(* CODESYS project BASIC.library
   Company: OSCAT
   DefaultNamespace: OSCAT_BASIC
   LanguageModelAttribute: qualified-access-only
   Title: BASIC
   Description: OSCAT Library with basic POUs.
      see www.oscat.de home of OSCAT library
   Author: OSCAT
   Version: 3.3.3.0

Project tree, tasks and I/O mapping:
  libraries: Standard, 3.5.2.0 (System)
  Data types/
    data type CALENDAR
    data type COMPLEX
    data type CONSTANTS_LANGUAGE
    data type CONSTANTS_LOCATION
    data type CONSTANTS_MATH
    data type CONSTANTS_PHYS
    data type CONSTANTS_SETUP
    data type ESR_DATA
    data type FRACTION
    data type HOLIDAY_DATA
    data type REAL2
    data type SDT
    data type TIMER_EVENT
    data type VECTOR_3
  Global Variables/
    global variables Constants
    global variables Globale_Variablen
    global variables Setup_Data
  POUs/
    Buffer Management/
      function _BUFFER_CLEAR [ST]
      function _BUFFER_INIT [ST]
      function _BUFFER_INSERT [ST]
      function _BUFFER_UPPERCASE [ST]
      function _STRING_TO_BUFFER [ST]
      function BUFFER_COMP [ST]
      function BUFFER_SEARCH [ST]
      function BUFFER_TO_STRING [ST]
    Engineering/
      automation/
        function block DRIVER_1 [ST]
        function block DRIVER_4 [ST]
        function block DRIVER_4C [ST]
        function block FLOW_CONTROL [ST]
        function block FT_Profile [ST]
        function block INC_DEC [ST]
        function block INTERLOCK [ST]
        function block INTERLOCK_4 [ST]
        function MANUAL [ST]
        function block MANUAL_1 [ST]
        function block MANUAL_2 [ST]
        function block MANUAL_4 [ST]
        function block PARSET [ST]
        function block PARSET2 [ST]
        function block SIGNAL [ST]
        function block SIGNAL_4 [ST]
        function block SRAMP [ST]
        function block TUNE [ST]
        function block TUNE2 [ST]
      control/
        function BAND_B [ST]
        function block CONTROL_SET1 [ST]
        function block CONTROL_SET2 [ST]
        function CTRL_IN [ST]
        function block CTRL_OUT [ST]
        function block CTRL_PI [ST]
        function block CTRL_PID [ST]
        function block CTRL_PWM [ST]
        function DEAD_BAND [ST]
        function block DEAD_BAND_A [ST]
        function DEAD_ZONE [ST]
        function block DEAD_ZONE2 [ST]
        function block FT_DERIV [ST]
        function block FT_IMP [ST]
        function block FT_INT [ST]
        function block FT_INT2 [ST]
        function block FT_PD [ST]
        function block FT_PDT1 [ST]
        function block FT_PI [ST]
        function block FT_PID [ST]
        function block FT_PIDW [ST]
        function block FT_PIDWL [ST]
        function block FT_PIW [ST]
        function block FT_PIWL [ST]
        function block FT_PT1 [ST]
        function block FT_PT2 [ST]
        function block FT_TN16 [ST]
        function block FT_TN64 [ST]
        function block FT_TN8 [ST]
        function block HYST [ST]
        function block HYST_1 [ST]
        function block HYST_2 [ST]
        function block HYST_3 [ST]
        function block INTEGRATE [ST]
      conversion/
        function block ASTRO [ST]
        function BFT_TO_MS [ST]
        function C_TO_F [ST]
        function C_TO_K [ST]
        function DEG_TO_DIR [ST]
        function DIR_TO_DEG [ST]
        function block ENERGY [ST]
        function F_TO_C [ST]
        function F_TO_OM [ST]
        function F_TO_PT [ST]
        function GEO_TO_DEG [ST]
        function K_TO_C [ST]
        function KMH_TO_MS [ST]
        function block LENGTH [ST]
        function MS_TO_BFT [ST]
        function MS_TO_KMH [ST]
        function OM_TO_F [ST]
        function block PRESSURE [ST]
        function PT_TO_F [ST]
        function block SPEED [ST]
        function block TEMPERATURE [ST]
      measurements/
        function block ALARM_2 [ST]
        function block BAR_GRAPH [ST]
        function block CALIBRATE [ST]
        function block CYCLE_TIME [ST]
        function block DT_SIMU [ST]
        function block FLOW_METER [ST]
        function block M_D [ST]
        function block M_T [ST]
        function block M_TX [ST]
        function block METER [ST]
        function block METER_STAT [ST]
        function block ONTIME [ST]
        function T_PLC_MS [ST]
        function T_PLC_US [ST]
        function block TC_MS [ST]
        function block TC_S [ST]
        function block TC_US [ST]
      sensor/
        function MULTI_IN [ST]
        function RES_NI [ST]
        function RES_NTC [ST]
        function RES_PT [ST]
        function RES_SI [ST]
        function SENSOR_INT [ST]
        function TEMP_NI [ST]
        function TEMP_NTC [ST]
        function TEMP_PT [ST]
        function TEMP_SI [ST]
      signal generators/
        function block _RMP_B [ST]
        function block _RMP_NEXT [ST]
        function block _RMP_W [ST]
        function block GEN_PULSE [ST]
        function block GEN_PW2 [ST]
        function block GEN_RDM [ST]
        function block GEN_RDT [ST]
        function block GEN_RMP [ST]
        function block GEN_SIN [ST]
        function block GEN_SQR [ST]
        function block PWM_DC [ST]
        function block PWM_PW [ST]
        function block RMP_B [ST]
        function block RMP_SOFT [ST]
        function block RMP_W [ST]
      signal processing/
        function AIN [ST]
        function block AIN1 [ST]
        function AOUT [ST]
        function AOUT1 [ST]
        function BYTE_TO_RANGE [ST]
        function block DELAY [ST]
        function block DELAY_4 [ST]
        function block FADE [ST]
        function block FILTER_DW [ST]
        function block FILTER_I [ST]
        function block FILTER_MAV_DW [ST]
        function block FILTER_MAV_W [ST]
        function block FILTER_W [ST]
        function block FILTER_WAV [ST]
        function MIX [ST]
        function MUX_R2 [ST]
        function MUX_R4 [ST]
        function OFFSET [ST]
        function OFFSET2 [ST]
        function OVERRIDE [ST]
        function RANGE_TO_BYTE [ST]
        function RANGE_TO_WORD [ST]
        function SCALE [ST]
        function SCALE_B [ST]
        function SCALE_B2 [ST]
        function SCALE_B4 [ST]
        function SCALE_B8 [ST]
        function SCALE_D [ST]
        function SCALE_R [ST]
        function SCALE_X2 [ST]
        function SCALE_X4 [ST]
        function SCALE_X8 [ST]
        function block SEL2_OF_3 [ST]
        function block SEL2_OF_3B [ST]
        function block SH [ST]
        function block SH_1 [ST]
        function block SH_2 [ST]
        function block SH_T [ST]
        function STAIR [ST]
        function block STAIR2 [ST]
        function block TREND [ST]
        function block TREND_DW [ST]
        function WORD_TO_RANGE [ST]
    List Processing/
      function LIST_ADD [ST]
      function LIST_CLEAN [ST]
      function LIST_GET [ST]
      function LIST_INSERT [ST]
      function LIST_LEN [ST]
      function block LIST_NEXT [ST]
      function LIST_RETRIEVE [ST]
      function LIST_RETRIEVE_LAST [ST]
    Logic/
      FF edge triggered/
        function block COUNT_BR [ST]
        function block COUNT_DR [ST]
        function block FF_D2E [ST]
        function block FF_D4E [ST]
        function block FF_DRE [ST]
        function block FF_JKE [ST]
        function block FF_RSE [ST]
        function block SELECT_8 [ST]
        function block SHR_4E [ST]
        function block SHR_4UDE [ST]
        function block SHR_8PLE [ST]
        function block SHR_8UDE [ST]
        function block TOGGLE [ST]
      FF pulse triggered/
        function block LTCH [ST]
        function block LTCH_4 [ST]
        function block STORE_8 [ST]
      gate logic/
        function BCDC_TO_INT [ST]
        function BIT_COUNT [ST]
        function BIT_LOAD_B [ST]
        function BIT_LOAD_B2 [ST]
        function BIT_LOAD_DW [ST]
        function BIT_LOAD_DW2 [ST]
        function BIT_LOAD_W [ST]
        function BIT_LOAD_W2 [ST]
        function BIT_OF_DWORD [ST]
        function BIT_TOGGLE_B [ST]
        function BIT_TOGGLE_DW [ST]
        function BIT_TOGGLE_W [ST]
        function BYTE_OF_BIT [ST]
        function BYTE_OF_DWORD [ST]
        function block BYTE_TO_BITS [ST]
        function BYTE_TO_GRAY [ST]
        function CHECK_PARITY [ST]
        function CHK_REAL [ST]
        function block DEC_2 [ST]
        function block DEC_4 [ST]
        function block DEC_8 [ST]
        function DW_TO_REAL [ST]
        function DWORD_OF_BYTE [ST]
        function DWORD_OF_WORD [ST]
        function GRAY_TO_BYTE [ST]
        function INT_TO_BCDC [ST]
        function MUX_2 [ST]
        function MUX_4 [ST]
        function PARITY [ST]
        function REAL_TO_DW [ST]
        function REFLECT [ST]
        function REVERSE [ST]
        function SHL1 [ST]
        function SHR1 [ST]
        function SWAP_BYTE [ST]
        function SWAP_BYTE2 [ST]
        function WORD_OF_BYTE [ST]
        function WORD_OF_DWORD [ST]
      generators/
        function block A_TRIG [ST]
        function block B_TRIG [ST]
        function block CLICK_CNT [ST]
        function block CLICK_DEC [ST]
        function block CLK_DIV [ST]
        function block CLK_N [ST]
        function block CLK_PRG [ST]
        function block CLK_PULSE [ST]
        function block CYCLE_4 [ST]
        function block D_TRIG [ST]
        function block GEN_BIT [ST]
        function block GEN_SQ [ST]
        function block SCHEDULER [ST]
        function block SCHEDULER_2 [ST]
        function block SEQUENCE_4 [ST]
        function block SEQUENCE_64 [ST]
        function block SEQUENCE_8 [ST]
        function block TMAX [ST]
        function block TMIN [ST]
        function block TOF_1 [ST]
        function block TONOF [ST]
        function block TP_1 [ST]
        function block TP_1D [ST]
        function block TP_X [ST]
      memory/
        function block FIFO_16 [ST]
        function block FIFO_32 [ST]
        function block STACK_16 [ST]
        function block STACK_32 [ST]
      Others/
        function CRC_GEN [ST]
        function block MATRIX [ST]
        function block PIN_CODE [ST]
    Mathematical/
      Array/
        function _ARRAY_ABS [ST]
        function _ARRAY_ADD [ST]
        function _ARRAY_INIT [ST]
        function _ARRAY_MEDIAN [ST]
        function _ARRAY_MUL [ST]
        function _ARRAY_SHUFFLE [ST]
        function _ARRAY_SORT [ST]
        function ARRAY_AVG [ST]
        function ARRAY_GAV [ST]
        function ARRAY_HAV [ST]
        function ARRAY_MAX [ST]
        function ARRAY_MIN [ST]
        function ARRAY_SDV [ST]
        function ARRAY_SPR [ST]
        function ARRAY_SUM [ST]
        function ARRAY_TREND [ST]
        function ARRAY_VAR [ST]
        function IS_SORTED [ST]
      Complex/
        function CABS [ST]
        function CACOS [ST]
        function CACOSH [ST]
        function CADD [ST]
        function CARG [ST]
        function CASIN [ST]
        function CASINH [ST]
        function CATAN [ST]
        function CATANH [ST]
        function CCON [ST]
        function CCOS [ST]
        function CCOSH [ST]
        function CDIV [ST]
        function CEXP [ST]
        function CINV [ST]
        function CLOG [ST]
        function CMUL [ST]
        function CPOL [ST]
        function CPOW [ST]
        function CSET [ST]
        function CSIN [ST]
        function CSINH [ST]
        function CSQRT [ST]
        function CSUB [ST]
        function CTAN [ST]
        function CTANH [ST]
      Double Precision/
        function R2_ABS [ST]
        function R2_ADD [ST]
        function R2_ADD2 [ST]
        function R2_MUL [ST]
        function R2_SET [ST]
      functions/
        function F_LIN [ST]
        function F_LIN2 [ST]
        function F_POLY [ST]
        function F_POWER [ST]
        function F_QUAD [ST]
        function FRMP_B [ST]
        function block FT_AVG [ST]
        function block FT_MIN_MAX [ST]
        function block FT_RMP [ST]
        function LINEAR_INT [ST]
        function POLYNOM_INT [ST]
      Geometry/
        function CIRCLE_A [ST]
        function CIRCLE_C [ST]
        function CIRCLE_SEG [ST]
        function CONE_V [ST]
        function ELLIPSE_A [ST]
        function ELLIPSE_C [ST]
        function SPHERE_V [ST]
        function TRIANGLE_A [ST]
      Vektormathematik/
        function V3_ABS [ST]
        function V3_ADD [ST]
        function V3_ANG [ST]
        function V3_DPRO [ST]
        function V3_NORM [ST]
        function V3_NUL [ST]
        function V3_PAR [ST]
        function V3_REV [ST]
        function V3_SMUL [ST]
        function V3_SUB [ST]
        function V3_XANG [ST]
        function V3_XPRO [ST]
        function V3_YANG [ST]
        function V3_ZANG [ST]
      function ACOSH [ST]
      function ACOTH [ST]
      function AGDF [ST]
      function ASINH [ST]
      function ATAN2 [ST]
      function ATANH [ST]
      function BETA [ST]
      function BINOM [ST]
      function CAUCHY [ST]
      function CAUCHYCD [ST]
      function CEIL [ST]
      function CEIL2 [ST]
      function CMP [ST]
      function COSH [ST]
      function COTH [ST]
      function D_TRUNC [ST]
      function DEC1 [ST]
      function DEG [ST]
      function DIFFER [ST]
      function ERF [ST]
      function ERFC [ST]
      function EVEN [ST]
      function EXP10 [ST]
      function EXPN [ST]
      function FACT [ST]
      function FIB [ST]
      function FLOOR [ST]
      function FLOOR2 [ST]
      function FRACT [ST]
      function GAMMA [ST]
      function GAUSS [ST]
      function GAUSSCD [ST]
      function GCD [ST]
      function GDF [ST]
      function GOLD [ST]
      function HYPOT [ST]
      function INC [ST]
      function INC1 [ST]
      function INC2 [ST]
      function INV [ST]
      function LAMBERT_W [ST]
      function LANGEVIN [ST]
      function MAX3 [ST]
      function MID3 [ST]
      function MIN3 [ST]
      function MODR [ST]
      function MUL_ADD [ST]
      function NEGX [ST]
      function RAD [ST]
      function RDM [ST]
      function RDM2 [ST]
      function RDMDW [ST]
      function REAL_TO_FRAC [ST]
      function RND [ST]
      function ROUND [ST]
      function SGN [ST]
      function SIGMOID [ST]
      function SIGN_I [ST]
      function SIGN_R [ST]
      function SINC [ST]
      function SINH [ST]
      function SQRTN [ST]
      function TANC [ST]
      function TANH [ST]
      function WINDOW [ST]
      function WINDOW2 [ST]
    Other/
      function block ESR_COLLECT [ST]
      function block ESR_MON_B8 [ST]
      function block ESR_MON_R4 [ST]
      function block ESR_MON_X8 [ST]
      function OSCAT_VERSION [ST]
      function STATUS_TO_ESR [ST]
    String/
      function BIN_TO_BYTE [ST]
      function BIN_TO_DWORD [ST]
      function BYTE_TO_STRB [ST]
      function BYTE_TO_STRH [ST]
      function CAPITALIZE [ST]
      function CHARCODE [ST]
      function CHARNAME [ST]
      function CHR_TO_STRING [ST]
      function CLEAN [ST]
      function CODE [ST]
      function COUNT_CHAR [ST]
      function COUNT_SUBSTRING [ST]
      function DEC_TO_BYTE [ST]
      function DEC_TO_DWORD [ST]
      function DEC_TO_INT [ST]
      function DEL_CHARS [ST]
      function DT_TO_STRF [ST]
      function DWORD_TO_STRB [ST]
      function DWORD_TO_STRF [ST]
      function DWORD_TO_STRH [ST]
      function EXEC [ST]
      function FILL [ST]
      function FIND_CHAR [ST]
      function FIND_CTRL [ST]
      function FIND_NONUM [ST]
      function FIND_NUM [ST]
      function FINDB [ST]
      function FINDB_NONUM [ST]
      function FINDB_NUM [ST]
      function FINDP [ST]
      function FIX [ST]
      function FLOAT_TO_REAL [ST]
      function FSTRING_TO_BYTE [ST]
      function FSTRING_TO_DT [ST]
      function FSTRING_TO_DWORD [ST]
      function FSTRING_TO_MONTH [ST]
      function FSTRING_TO_WEEK [ST]
      function FSTRING_TO_WEEKDAY [ST]
      function HEX_TO_BYTE [ST]
      function HEX_TO_DWORD [ST]
      function IS_ALNUM [ST]
      function IS_ALPHA [ST]
      function IS_CC [ST]
      function IS_CTRL [ST]
      function IS_HEX [ST]
      function IS_LOWER [ST]
      function IS_NCC [ST]
      function IS_NUM [ST]
      function IS_UPPER [ST]
      function ISC_ALPHA [ST]
      function ISC_CTRL [ST]
      function ISC_HEX [ST]
      function ISC_LOWER [ST]
      function ISC_NUM [ST]
      function ISC_UPPER [ST]
      function LOWERCASE [ST]
      function block MESSAGE_4R [ST]
      function block MESSAGE_8 [ST]
      function MIRROR [ST]
      function MONTH_TO_STRING [ST]
      function OCT_TO_BYTE [ST]
      function OCT_TO_DWORD [ST]
      function REAL_TO_STRF [ST]
      function REPLACE_ALL [ST]
      function REPLACE_CHARS [ST]
      function REPLACE_UML [ST]
      function block TICKER [ST]
      function TO_LOWER [ST]
      function TO_UML [ST]
      function TO_UPPER [ST]
      function TRIM [ST]
      function TRIM1 [ST]
      function TRIME [ST]
      function UPPERCASE [ST]
      function WEEKDAY_TO_STRING [ST]
      function LREAL_TO_STRF [ST]
    Time&Date/
      function block CALENDAR_CALC [ST]
      function DATE_ADD [ST]
      function DAY_OF_DATE [ST]
      function DAY_OF_MONTH [ST]
      function DAY_OF_WEEK [ST]
      function DAY_OF_YEAR [ST]
      function DAY_TO_TIME [ST]
      function DAYS_DELTA [ST]
      function DAYS_IN_MONTH [ST]
      function DAYS_IN_YEAR [ST]
      function block DCF77 [ST]
      function DST [ST]
      function DT2_TO_SDT [ST]
      function DT_TO_SDT [ST]
      function EASTER [ST]
      function block EVENTS [ST]
      function block HOLIDAY [ST]
      function HOUR [ST]
      function HOUR_OF_DT [ST]
      function HOUR_TO_TIME [ST]
      function HOUR_TO_TOD [ST]
      function JD2000 [ST]
      function LEAP_DAY [ST]
      function LEAP_OF_DATE [ST]
      function LEAP_YEAR [ST]
      function LTIME_TO_UTC [ST]
      function MINUTE [ST]
      function MINUTE_OF_DT [ST]
      function MINUTE_TO_TIME [ST]
      function MONTH_BEGIN [ST]
      function MONTH_END [ST]
      function MONTH_OF_DATE [ST]
      function MULTIME [ST]
      function PERIOD [ST]
      function PERIOD2 [ST]
      function REFRACTION [ST]
      function block RTC_2 [ST]
      function block RTC_MS [ST]
      function SDT_TO_DATE [ST]
      function SDT_TO_DT [ST]
      function SDT_TO_TOD [ST]
      function SECOND [ST]
      function SECOND_OF_DT [ST]
      function SECOND_TO_TIME [ST]
      function SET_DATE [ST]
      function SET_DT [ST]
      function SET_TOD [ST]
      function SUN_MIDDAY [ST]
      function block SUN_POS [ST]
      function block SUN_TIME [ST]
      function TIMECHECK [ST]
      function UTC_TO_LTIME [ST]
      function WORK_WEEK [ST]
      function YEAR_BEGIN [ST]
      function YEAR_END [ST]
      function YEAR_OF_DATE [ST]
*)

// Data types/CALENDAR
TYPE CALENDAR :
STRUCT
	UTC : DT;					(* world time UTC *)
	_LDT : DT;					(* local time *)
	_LDATE : DATE;				(* local date *)
	_LTOD : TOD;					(* local time of day *)
	YEAR : INT;					(* year of LDATE *)
	MONTH : INT;				(* month of LDATE *)
	DAY : INT;					(* day of LDATE *)
	WEEKDAY : INT;				(* weekday of LDATE *)
	OFFSET : INT;				(* Time Zone Offset for Local time in minutes *)
	DST_EN : BOOL;				(* daylight savings time enable *)
	DST_ON : BOOL;				(* true when daylight savings time os on *)
	NAME : STRING(5);			(* name of time zone *)
	LANGUAGE : INT;			(* location number pls see location setup *)
	LONGITUDE : REAL;			(* longitude of current location *)
	LATITUDE : REAL;			(* latitude of current location *)
	SUN_RISE : TOD;				(* sun_rise for current location *)
	SUN_SET : TOD;				(* sun_set for current location *)
	SUN_MIDDAY : TOD;			(* worldtime when sun stands at south position *)
	SUN_HEIGTH : REAL	;		(* suns heigth at midday, south position *)
	SUN_HOR : REAL;			(* sun angle horizontal 0 = north in degrees *)
	SUN_VER : REAL;			(* sun angle vertical above horizon in degrees *)
	NIGHT : BOOL;				(* true between sun_set and sun_rise *)
	HOLIDAY : BOOL;			(* true when holiday *)
	HOLY_NAME : STRING(30);	(* name of holiday *)
	WORK_WEEK : INT;			(* current work week *)
END_STRUCT
END_TYPE

// Data types/COMPLEX
TYPE COMPLEX :
STRUCT
	re : REAL;
	im : REAL;
END_STRUCT
END_TYPE

// Data types/CONSTANTS_LANGUAGE
TYPE CONSTANTS_LANGUAGE :
STRUCT
	(* Language Setup *)
	DEFAULT : INT := 1; (* 1=english, 2=german 3=french *)
	LMAX : INT := 3;
	WEEKDAYS : ARRAY[1..3, 1..7] OF STRING(10) :=[	'Monday', 'Tuesday', 'Wednesday', 'Thursday', 'Friday', 'Saturday', 'Sunday',
													'Montag', 'Dienstag', 'Mittwoch', 'Donnerstag', 'Freitag', 'Samstag', 'Sonntag',
													'Lundi', 'Mardi', 'Mercredi', 'Jeudi', 'Vendredi', 'Samedi', 'Dimanche'];
	WEEKDAYS2 : ARRAY[1..3, 1..7] OF STRING(2) :=[	'Mo', 'Tu', 'We', 'Th', 'Fr', 'Sa', 'Su',
													'Mo', 'Di', 'Mi', 'Do', 'Fr', 'Sa', 'So',
													'Lu', 'Ma', 'Me', 'Je', 'Ve', 'Sa', 'Di'];
	MONTHS : ARRAY[1..3, 1..12] OF STRING(10) :=[	'January', 'February', 'March', 'April', 'May', 'June', 'July', 'August', 'September', 'October', 'November', 'December',
													'Januar', 'Februar', 'März', 'April', 'Mai', 'Juni', 'Juli', 'August', 'September', 'Oktober', 'November', 'Dezember',
													'Janvier', 'Février', 'mars', 'Avril', 'Mai', 'Juin', 'Juillet', 'Août', 'Septembre', 'Octobre', 'Novembre', 'Decembre'];
	MONTHS3 : ARRAY[1..3, 1..12] OF STRING(3) :=[	'Jan', 'Feb', 'Mar', 'Apr', 'May', 'Jun', 'Jul', 'Aug', 'Sep', 'Oct', 'Nov', 'Dec',
													'Jan', 'Feb', 'Mrz', 'Apr', 'Mai', 'Jun', 'Jul', 'Aug', 'Sep', 'Okt', 'Nov', 'Dez',
													'Jan', 'Fev', 'Mar', 'Avr', 'Mai', 'Jun', 'Jul', 'Aou', 'Sep', 'Oct', 'Nov', 'Dec'];
	DIRS : ARRAY[1..3,0..15] OF STRING(3) :=[		'N', 'NNE', 'NE', 'ENE', 'E', 'ESE', 'SE', 'SSE', 'S', 'SSW', 'SW', 'WSW', 'W', 'WNW', 'NW', 'NNW',
													'N', 'NNO', 'NO', 'ONO', 'O', 'OSO', 'SO', 'SSO', 'S', 'SSW', 'SW', 'WSW', 'W', 'WNW', 'NW', 'NNW',
													'N', 'NNO', 'NO', 'ONO', 'O', 'OSO', 'SO', 'SSO', 'S', 'SSW', 'SW', 'WSW', 'W', 'WNW', 'NW', 'NNW'];
END_STRUCT
END_TYPE

// Data types/CONSTANTS_LOCATION
TYPE CONSTANTS_LOCATION :
STRUCT
	(* location setup *)
	DEFAULT : INT := 1; (* 1=germany, 2=austria 3=france 4=belgium-german 5= italien-Südtirol *)
	LMAX : INT := 5;

	(* language spoken in the location *)
	LANGUAGE : ARRAY[1..5] OF INT :=[ 2, 2, 3, 2, 2];

END_STRUCT
END_TYPE

// Data types/CONSTANTS_MATH
TYPE CONSTANTS_MATH :
STRUCT
	PI : REAL := 	3.14159265358979323846264338327950288;		(* Kreiszahl PI *)
	PI2 : REAL := 	6.28318530717958647692528676655900576;	(* PI * 2 *)
	PI4 : REAL :=  12.56637061435917295385057353311801152;	(* PI * 4 *)
	PI05 : REAL :=  1.5707963267949;							(* PI / 2 *)
	PI025 : REAL := 0.785398163397448;							(* PI / 4 *)
	PI_INV : REAL := 0.318309886183791;						(* 1 / PI *)
	E : REAL := 	2.71828182845904523536028747135266249;		(* Euler constant e *)
	E_INV : REAL := 0.367879441171442;							(* 1 / e *)
	SQ2 : REAL :=	1.4142135623731;							(* Wurzel von 2 *)
	FACTS : ARRAY[0..12] OF DINT :=[ 1,1,2,6,24,120,720,5040,40320,362880,3628800,39916800,479001600];
END_STRUCT
END_TYPE

// Data types/CONSTANTS_PHYS
TYPE CONSTANTS_PHYS :
STRUCT
	C : REAL := 299792458.0;				(* Lichtgeschwindigkeit in m/s *)
	E : REAL := 1.60217653E-19;				(* elementarladung in Colomb = A * s *)
	G : REAL := 9.80665; 						(* Erdbeschleunigung in m / s² *)
	T0 : REAL := -273.15;						(* absoluter Nullpunkt in °C *)
	RU : REAL := 8.314472; 					(* Universelle Gaskonstante in J / (mol · K) *)
	PN : REAL := 101325.0;					(* NormalDruck in Pa *)
END_STRUCT
END_TYPE

// Data types/CONSTANTS_SETUP
TYPE CONSTANTS_SETUP :
STRUCT
	(* setup Parameters *)
	EXTENDED_ASCII : BOOL := TRUE;
	CHARNAMES : ARRAY[1..4] OF STRING(253) :=[ ';"&quot;&&amp;<&lt;>&gt;€&euro; &nbsp;¡&iexcl;¢&cent;£&pound;¤&curren;¥&yen;¦&brvbar;§&sect;¨&uml;©&copy;ª&ordf;«&laquo;¬&not;­&shy;®&reg;¯&macr;°&deg;±&plusmn;²&sup2;³&sup3;´&acute;µ&micro;¶&para;·&middot;¸&cedil;¹&sup1;º&ordm;»&raquo;¼&frac14;Û&Ucirc;',
		';¾&frac34;¿&iquest;À&Agrave;Á&Aacute;Â&Acirc;Ã&Atilde;Ä&Auml;Å&Aring;Æ&AElig;Ç&Ccedil;È&Egrave;É&Eacute;Ê&Ecirc;Ë&Euml;Ì&Igrave;Í&Iacute;Î&Icirc;Ï&Iuml;Ð&ETH;Ñ&Ntilde;Ò&Ograve;Ó&Oacute;Ô&Ocirc;Õ&Otilde;Ö&Ouml;×&times;Ø&Oslash;Ù&Ugrave;Ú&Uacute;½&frac12;',
		';Ü&Uuml;Ý&Yacute;Þ&THORN;ß&szlig;à&agrave;á&aacute;â&acirc;ã&atilde;ä&auml;å&aring;æ&aelig;ç&ccedil;è&egrave;é&eacute;ê&ecirc;ë&euml;ì&igrave;í&iacute;î&icirc;ï&iuml;ð&eth;ñ&ntilde;ò&ograve;ó&oacute;ô&ocirc;õ&otilde;ö&ouml;÷&divide;ø&oslash;ù&ugrave;',
		';ú&uacute;û&ucirc;ü&uuml;ý&yacute;þ&thorn;ÿ&yuml;'];
	MTH_OFS : ARRAY[1..12] OF INT :=[ 0,31,59,90,120,151,181,212,243,273,304,334];
	DECADES : ARRAY[0..8] OF REAL :=[ 1.0,10.0,100.0,1000.0,10000.0,10000.0,100000.0,1000000.0,10000000.0];
END_STRUCT
END_TYPE

// Data types/ESR_DATA
TYPE ESR_DATA :
STRUCT
	TYP : BYTE;
	ADRESS : STRING(10);
	DS : DT;
	TS : TIME;
	DATA : ARRAY[0..7] OF BYTE;
END_STRUCT
END_TYPE

// Data types/FRACTION
TYPE FRACTION :
STRUCT
	NUMERATOR : INT;
	DENOMINATOR : INT;
END_STRUCT
END_TYPE

// Data types/HOLIDAY_DATA
TYPE HOLIDAY_DATA :
STRUCT
	NAME : STRING(30);
	DAY : SINT;
	MONTH : SINT;
	USE : SINT;
END_STRUCT
END_TYPE

// Data types/REAL2
TYPE REAL2 :
STRUCT
	R1 : REAL;	(* small value *)
	RX : REAL;	(* big value *)
END_STRUCT
END_TYPE

// Data types/SDT
TYPE SDT :
STRUCT
	YEAR : INT;
	MONTH : INT;
	DAY : INT;
	WEEKDAY : INT;
	HOUR : INT;
	MINUTE : INT;
	SECOND : INT;
	MS : INT;
END_STRUCT
END_TYPE

// Data types/TIMER_EVENT
TYPE TIMER_EVENT :
STRUCT
	TYP : BYTE;
	CHANNEL : BYTE;
	DAY : BYTE;
	START : TOD;
	DURATION : TIME;
	LAND : BYTE;
	LOR : BYTE;
	LAST : DT;
END_STRUCT
END_TYPE

// Data types/VECTOR_3
TYPE VECTOR_3 :
STRUCT
	X : REAL;
	Y : REAL;
	Z : REAL;
END_STRUCT
END_TYPE

// Global Variables/Constants
VAR_GLOBAL CONSTANT
	STRING_LENGTH : INT := 250;
	LIST_LENGTH : INT := 250;
END_VAR




(* revisionhistory
hm 3. mar. 2007
	extended accuracy of pi2
	renamed T0 to Tk for better compatibility with other libraries
	renamed C t0 c0 for better compatibility

hm	2. may. 2007
	added RU universal gas constant

hm	1. oct. 2007
	added setup parameter STEP7

hm 31. oct. 2007
	added PN

hm	6. mar. 2008
	added setup Parameter EXTENDED_ASCII

hm	28. Mar. 2008
	added setup parameter STRING_LENGTH

hm	7. apr. 2008
	Deleted unused setup parameter Step7

hm	19. apr. 2008
	added setup parameter NETWORK_BUFFER_SIZE

hm	27. apr. 2008
	added PI05 and PI025

hm	18. may. 2008
	added charname lists
	renamed E to E1

hm	30. jun. 2008
	reduced size of string constants to 253 to avoid problems with target aixia DCUF

hm	21. sep. 2008
	added section language setup
	added section location setup

hm	20. oct. 2008
	changed to structured constants

hm	16. nov. 2008
	moved structured constants to global vars for compatibility reasons

hm	13. nov. 2009
	added network_buffer_short_size
	renamed network_buffer_long_size
	changed string length to 250

hm	20. jan. 2011
	removed network buffers
	added list_length
*)

// Global Variables/Globale_Variablen
VAR_GLOBAL
	MATH : CONSTANTS_MATH;
	PHYS : CONSTANTS_PHYS;
	LANGUAGE : CONSTANTS_LANGUAGE;
	SETUP : CONSTANTS_SETUP;
	LOCATION : CONSTANTS_LOCATION;
END_VAR

// Global Variables/Setup_Data
VAR_GLOBAL RETAIN

END_VAR

// POUs/Mathematical/Array/_ARRAY_ABS
FUNCTION _ARRAY_ABS : BOOL
VAR_INPUT
	pt : POINTER TO ARRAY[0..32000] OF REAL;
	size : UINT;
END_VAR
VAR
	i: UINT;
	stop: UINT;
END_VAR

(*
version 1.0	2. apr. 2008
programmer 	hugo
tested by	tobias

this function will calculate the absolute value of each element of the array and stroe the result instead of the element.
Array[i] := ABS(ARRAY[i]).
the function needs to be called:	array_avg(adr("array"),sizeof("array"));
because this function works with pointers its very time efficient and it needs no extra memory.

*)

stop := SHR(size,2)-1;
FOR i := 0 TO stop DO
	PT^[i] := ABS(PT^[i]);
END_FOR;
_ARRAY_ABS := TRUE;


(* revision history
hm	2. apr 2008		rev 1.0
	original version

*)

END_FUNCTION

// POUs/Mathematical/Array/ARRAY_AVG
FUNCTION ARRAY_AVG : REAL
VAR_INPUT
	pt : POINTER TO ARRAY[0..32000] OF REAL;
	size : UINT;
END_VAR
VAR
	i: UINT;
	stop: UINT;
END_VAR

(*
version 1.3	10. mar. 2009
programmer 	hugo
tested by		tobias

this function will calculate the average of a given array.
the function needs to be called:	array_avg(adr("array"),sizeof("array"));
because this function works with pointers its very time efficient and it needs no extra memory.

*)

stop := SHR(size,2)-1;
ARRAY_AVG := pt^[0];
FOR i := 1 TO stop DO
	ARRAY_AVG := ARRAY_AVG + pt^[i];
END_FOR;
ARRAY_AVG := ARRAY_AVG / UINT_TO_REAL(stop + 1);


(* revision history
hm	2. oct 2007		rev 1.0
	original version

hm	12. dec 2007	rev 1.1
	chaged code for better performance

hm	16. mar. 2008	rev 1.2
	changed input size to uint

hm	10. mar. 2009	rev 1.3
	added type conversion for compatibility reasons
*)

END_FUNCTION

// POUs/String/CODE
FUNCTION CODE : BYTE
VAR_INPUT
	STR : STRING(STRING_LENGTH);
	POS : INT;
END_VAR
VAR
	PT : POINTER TO BYTE;
END_VAR

(*
version 1.1	29. mar. 2008
programmer 	hugo
tested by		tobias

code extracts the code of a character at position POS of a string STR.

*)

IF pos < 1 OR pos > LEN(str) THEN
	CODE := 0;
	RETURN;
ELSE
	PT := ADR(STR) + INT_TO_DWORD(pos - 1);
	CODE := pt^;
END_IF;

(* revision history
hm	9. mar. 2008	rev 1.0
	original version

hm	29. mar. 2008	rev 1.1
	changed STRING to STRING(STRING_LENGTH)
*)

END_FUNCTION

// POUs/Mathematical/Array/_ARRAY_ADD
FUNCTION _ARRAY_ADD : BOOL
VAR_INPUT
	pt : POINTER TO ARRAY[0..32000] OF REAL;
	size : UINT;
	X : REAL;
END_VAR
VAR
	i: UINT;
	stop: UINT;
END_VAR

(*
version 1.0	2. apr. 2008
programmer 	hugo
tested by	tobias

this function will add an offset X to each element of the array and stroe the result instead of the element.
Array[i] := ARRAY[i] + X.
the function needs to be called:	array_avg(adr("array"),sizeof("array"));
because this function works with pointers its very time efficient and it needs no extra memory.

*)

stop := SHR(size,2)-1;
FOR i := 0 TO stop DO
	PT^[i] := PT^[i] + X;
END_FOR;
_ARRAY_ADD := TRUE;


(* revision history
hm	2. apr 2008		rev 1.0
	original version

*)

END_FUNCTION

// POUs/Engineering/signal processing/OFFSET
FUNCTION OFFSET : REAL
VAR_INPUT
	X : REAL;
	O1, O2, O3, O4 : BOOL;
	D : BOOL;
END_VAR
VAR_INPUT CONSTANT
	Offset_1 : REAL;
	Offset_2 : REAL;
	Offset_3 : REAL;
	Offset_4 : REAL;
	default : REAL;
END_VAR

(*
version 1.0	12 jan 2007
programmer 	oscat
tested by	oscat

The Function offset adds offsets to an analog signal depending on digital inputs.
all selected offsets are added at the same time.
with the input D a default value instead of the input X can be used.

*)

IF D THEN OFFSET := default; ELSE OFFSET := X; END_IF;
IF O1 THEN OFFSET := OFFSET + offset_1; END_IF;
IF O2 THEN OFFSET := OFFSET + offset_2; END_IF;
IF O3 THEN OFFSET := OFFSET + offset_3; END_IF;
IF O4 THEN OFFSET := OFFSET + offset_4; END_IF;



(* revision history
hm	12. jan 2007
	original version


*)

END_FUNCTION

// POUs/Engineering/automation/SIGNAL
FUNCTION_BLOCK SIGNAL
VAR_INPUT
	IN : BOOL;
	SIG : BYTE;
	TS : TIME;
END_VAR
VAR_OUTPUT
	Q : BOOL;
END_VAR
VAR
	tx: DWORD;
	step: BYTE;
END_VAR
VAR CONSTANT
	one : BYTE := 1;
END_VAR

(*
version 1.0	13 dec 2007
programmer 	hugo
tested by		tobias

this function generates an output signal according to a bit pattern SIG.
the patter is shifted to the output in time steps of TS.
ts defaults to 128 ms if not specified.
*)

IF in THEN
	(* an alarm is present read system time first *)
	tx := T_PLC_MS();
	(* calculate the step counter which is the lowest 3 bits of (time / ts) *)
	IF ts > t#0s THEN
		step := DWORD_TO_BYTE(tx / TIME_TO_DWORD(ts) AND 16#0000_0007);
	ELSE
		step := DWORD_TO_BYTE(SHR(tx,7) AND 16#0000_0007);
	END_IF;
	(* convert the value 0-7 in step into one bit only (bit 0-7) *)
	step := SHL(one,step);
	(* generate the output signal *)
	Q := (step AND sig) > 0;
ELSE
	Q := FALSE;
END_IF;

(* revision history
hm	13.12.2007		rev 1.0
	original version

*)

END_FUNCTION_BLOCK

// POUs/Engineering/measurements/T_PLC_MS
FUNCTION T_PLC_MS : DWORD
VAR CONSTANT
	debug : BOOL := 0;
	N : INT := 0;
	offset : DWORD := 0;
END_VAR
VAR
	tx : TIME;
END_VAR

(*
version 1.2	16. nov 2008
programmer 	hugo
tested by	oscat

T_PLC_MS reads the internal PLC timer and return the time, it has the advantage to be able to set a debug mode 
and speed up the counter to test the plc timer overrun which occurs every 50 days respectively 25 days at siemens S7
this routine also allows to correct the behavior of s7 where the internal plc counter will not count all 32 bits.

*)

tx := TIME();
T_PLC_MS := TIME_TO_DWORD(Tx);
(* hier muss die korrektur für step7 stattfinden
plctime muss den vollen wertebereich von time ausnutzen:
wenn bei step7 time -24tage bis plus 24 tage ist dann muss der timer auch beim überlauf auf -24tage springen 
und auf keinen fall auf 0 !!!!
für siemens muss ein weiterer fb im main eingebunden werden der sicherstellt das alle 32 bits durchgezählt werden.
es kann nur ein fb sein den er muss sich das oberste (32te) bit merken.
oder etwa spring s7 bei überlauf auf -24 tage????? dann wäre keine korrektur nötig.
*)
IF debug THEN
	T_PLC_MS := (SHL(T_PLC_MS,N) OR SHL(DWORD#1,N)-1) + OFFSET;
END_IF;

(* revision history
hm	14.9.2007	rev 1.0
	original version

hm	12. nov 2007	rev 1.1
	added temporaray variable tx because some compilers could not handle time() as an argument

hm	16. nov. 2008	rev 1.2
	initialized constants with 0 for compatibility reasons
*)

END_FUNCTION

// POUs/Engineering/conversion/SPEED
FUNCTION_BLOCK SPEED
VAR_INPUT
	ms : REAL;
	kmh : REAL;
	kn : REAL;
	mh : REAL;
END_VAR
VAR_OUTPUT
	Yms : REAL;
	Ykmh : REAL;
	Ykn : REAL;
	Ymh : REAL;
END_VAR


(*
version 1.1	11. mar. 2009
programmer 	hugo
tested by		oscat

this function converts different speed units
any unused input can simply be left open.
different inputs connected at the same time will be added up.

*)

Yms := ms +
		kmh * 0.27777777777778 +
		kn * 0.5144444 +
		mh * 0.44704;
Ykmh := Yms * 3.6;
Ykn := Yms * 1.94384466037535;
Ymh := Yms * 2.23693629205440;

(*
Geschwindigkeit Meter durch Sekunde m/s 1 m/s = 3,6 km/h
km durch (pro) Stunde, nicht „Stundenkilometer“ verwenden
Knoten kn 1 kn = 1 sm/h = 0,5144 m/s

*)

(* revision history
hm	27. mar. 2009	rev 1.0
	original version

hm	11. mar. 2009	rev 1.1
	improved code

*)

END_FUNCTION_BLOCK

// POUs/Engineering/measurements/METER
FUNCTION_BLOCK METER
VAR_INPUT
	M1, M2 : REAL;
	I1, I2 : BOOL;
	D : REAL := 1.0;
	RST : BOOL;
END_VAR
VAR_IN_OUT
	MX : REAL;
END_VAR
VAR
	MR : REAL2;
	MX1, MX2 : REAL; (* current consumption value on M1 and M2 *)
	tx: DWORD;
	last: DWORD;
	tc: REAL;
	init: BOOL;
END_VAR

(*
	version 1.4	8. mar. 2009
	programmer 	oscat
	tested BY	oscat

METER measures usage of power or similar values the output MX is the sum of the inputs over time.
MX := sum over time of (I1 * P1 + I2 * P2)/D.
a simple example is the consumption counter for a 2 stage oil burner where stage 1 is 10KW and stage 2 is 20KW.
I1 and I2 decide which value is accounted for, I1 = True only counts P1, I2 is True counts P2 
and I1 and I2 is true counts P1 and P2.
the meter can be used for all kind of consumption meters. P1 and P2 can change on the fly.

*)

(* measure the last cycle time and make sure we onle execute once every millisecond *)
tx := T_PLC_MS();
IF NOT init THEN
	init := TRUE;
	last := tx;
	mr.RX := mx;
	mr.R1 := 0.0;
ELSIF tx = last THEN
	RETURN;
ELSE
	tc := DWORD_TO_REAL(tx - last) * 0.001;
END_IF;
last := tx;

(* reset *)
IF rst THEN
	mr.R1 := 0.0;
	mr.RX := 0.0;
ELSE
	(* current consumption measurement *)
	IF I1 THEN MX1 := M1; ELSE MX1 := 0.0; END_IF;
	IF I2 THEN MX2 := M2; ELSE MX2 := 0.0; END_IF;
	(* add up the current values in a double real *)
	MR := R2_ADD(MR,(SEL(I1,0.0,mx1) + SEL(I2, 0.0, mx2)) / D * TC);
	(* set the current output value *)
	MX := mr.RX;
END_IF;




(* revision history

hm	16. sep.2007		rev 1.0
	original version

hm	7. feb 2008		rev 1.1
	use new version of ft_int to avoid a counting stop at high values
	deleted unnecessary limits

hm	24. mar. 2008	rev 1.2
	use data_type real2 to extend accuracy to 15 digits total
	do not use ft_int which adds unnecessary overhead

hm	8. feb. 2009	rev 1.3
	changed mx to be I/O
	make sure calculation works for cycle times < 1 ms

hm	8. mar. 2009	rev 1.4
	last was not updated
	code improvements

*)

END_FUNCTION_BLOCK

// POUs/Mathematical/Double Precision/R2_ADD
FUNCTION R2_ADD : REAL2
VAR_INPUT
	X : Real2;
	Y : REAL;
END_VAR
VAR
	temp: REAL;
END_VAR

(*
version 1.0	20. mar. 2008
programmer 	hugo
tested by	tobias

R2_add adds a real to a double real which extends the accuracy of a real to twice as many digits

*)

temp := X.RX;
R2_ADD.RX := Y + X.R1 + X.RX;
R2_ADD.R1 := temp - R2_ADD.RX + Y + X.R1;


(* revision history
hm		20.3.2008	rev 1.0
	original version

*)

END_FUNCTION

// POUs/Engineering/control/FT_INT
FUNCTION_BLOCK FT_INT
VAR_INPUT
	IN : REAL;
	K : REAL := 1;
	RUN : BOOL := TRUE;
	RST : BOOL;
	OUT_MIN : REAL := -1E37;
	OUT_MAX : REAL := 1E37;
END_VAR
VAR_OUTPUT
	OUT : REAL;
	LIM : BOOL;
END_VAR
VAR
	INTeg : INTEGRATE;
END_VAR


(*
version 2.2	10. mar. 2009
programmer 	hugo
tested by		oscat

FT_int is an integrator with input IN and factor K.
integration is only done while run = true, if run is false integration is stopped and the out remains at the last value.
if run is left unconnected, run is considered true by the function block.
the output ET will display the total integration time from last reset.
the out_min and out_max values can be set to ,imit the output value range. 
the default for K is 1.

 
*)

IF rst THEN
	out := 0.0;
ELSE
	integ(X := IN, E := RUN, K := K, Y := out);
END_IF;

(* limit the outputs *)
IF out >= OUT_MAX THEN
	out := out_max;
	LIM := TRUE;
ELSIF out <= out_min THEN
	out := out_min;
	lim := TRUE;
ELSE
	lim := FALSE;
END_IF;


(*
hm 13.12.2006	rev 1.1
	changed to "trapezregel" which increases accuracy
	before out := out + in * time new: out := out + (in + in_last) / 2 * time

hm 15.1.2007		rev 1.2
	added default for k to be 1.

hm	15.9.2007		rev 1.3
	replaced time() with T_PLC_US for compatibility and performance reason
	increased internal accuracy to microseconds

hm 29. oct 2007		rev 1.4
	changed code so int will not be called is time difference is 0 to increase accuracy on systems
	with cycle times below 1ms

hm	2. dec 2007	 	rev 1.5
	changed code for better performance

hm	5. jan 2008		rev 1.6
	further improvements in performance

hm	8. feb 2008		rev 1.7
	deleted limits +/- 1000 now limit is the range of real
	added variables out1 and out2 to extend the resolution
	corrected an error with elapsed time
	deleted unusfull output ET

hm	13. mar 2008	rev 1.8
	changed preset value out_min to -1e37.
	stop integrator at the limits.

hm	16. mar 2008	rev 1.9
	added type conversion to avoid warning under codesys 3.0

hm	2. jun. 2008	rev 2.0
	rewritten with clear code
	limits can now be set without run

hm	3. nov. 2008	rev 2.1
	optimized code using INTEGRATE and LIMX

hm	10. mar. 2009	rev 2.2
	removed nested comments
*)

END_FUNCTION_BLOCK

// POUs/Engineering/measurements/T_PLC_US
FUNCTION T_PLC_US : DWORD
VAR CONSTANT
	debug : BOOL := 0;
	N : INT := 0;
	offset : DWORD := 0;
END_VAR
VAR
	tx : TIME;
END_VAR

(*
version 1.2	16 nov 2008
programmer 	hugo
tested by	tobias

T_PLC_US reads the internal PLC timer and return the time, it has the advantage to be able to set a debug mode 
and speed up the counter to test the plc timer overrun which occurs every 50 days respectively 25 days at siemens S7
this routine also allows to correct the behavior of s7 where the internal plc counter will not count all 32 bits.

*)

tx := TIME();
T_PLC_US := TIME_TO_DWORD(Tx)*1000;
(* hier muss die korrektur für step7 stattfinden
plctime muss den vollen wertebereich von time ausnutzen:
wenn bei step7 time -24tage bis plus 24 tage ist dann muss der timer auch beim überlauf auf -24tage springen 
und auf keinen fall auf 0 !!!!
für siemens muss ein weiterer fb im main eingebunden werden der sicherstellt das alle 32 bits durchgezählt werden.
es kann nur ein fb sein den er muss sich das oberste (32te) bit merken.
oder etwa spring s7 bei überlauf auf -24 tage????? dann wäre keine korrektur nötig.
*)
IF debug THEN
	T_PLC_US := (SHL(T_PLC_US,N) OR SHL(DWORD#1,N)-1) + OFFSET;
END_IF;

(* revision history
hm	14.9.2007	rev 1.0
	original version

hm	12. nov 2007	rev 1.1
	added temporaray variable tx because some compilers could not handle time() as an argument

hm	16. nov. 2008	rev 1.2
	initialized constants with 0 for compatibility reasons

*)

END_FUNCTION

// POUs/Engineering/control/INTEGRATE
FUNCTION_BLOCK INTEGRATE
VAR_INPUT
	E : BOOL := TRUE;
	X : REAL;
	K : REAL := 1.0;
END_VAR
VAR_IN_OUT
	Y : REAL;
END_VAR
VAR
	X_last : REAL;
	init: BOOL;
	last: DWORD;
	tx: DWORD;
END_VAR


(*
version 1.0	3. nov. 2008
programmer 	hugo
tested by	oscat

integrate is a plain integrator with I/O for out.

 
*)

(*read system time *)
tx := T_PLC_MS();

IF NOT init THEN
	init := TRUE;
	X_last := X;
ELSIF E THEN
	Y := (X + X_LAST) * 0.5E-3 * DWORD_TO_REAL(tx-last) * K + Y;
	X_last := X;
END_IF;
last := tx;



(*
hm 3. nov. 2008	rev 1.0
original version
	
*)

END_FUNCTION_BLOCK

// POUs/Mathematical/Array/_ARRAY_INIT
FUNCTION _ARRAY_INIT : BOOL
VAR_INPUT
	pt : POINTER TO ARRAY[0..32000] OF REAL;
	size : UINT;
	init : REAL;
END_VAR
VAR
	i: UINT;
	stop: UINT;
END_VAR


(*
version 1.3	16 mar 2008
programmer 	hugo
tested by		tobias

this function will initialize a given array with a value init.
the function needs to be called:	_array_init(adr("array"),sizeof("array"));
this function will manipulate a given array.
the function manipulates the original array, it rerturnes true when finished.
because this function works with pointers its very time efficient and it needs no extra memory.

*)

stop := SHR(size,2)-1;
FOR i := 0 TO stop DO
	pt^[i] := init;
END_FOR;

_array_init := TRUE;

(* revision History

hm 6.1.2007		rev 1.1
	change type of function to bool
	added  array_init := true to set output true.

hm	14.11.2007	rev 1.2
	changed stop calculation to be more efficient

hm	16.3. 2008		rev 1.3
	changed type of input size to uint
*)

END_FUNCTION

// POUs/Mathematical/Array/_ARRAY_MEDIAN
FUNCTION _ARRAY_MEDIAN : REAL
VAR_INPUT
	pt : POINTER TO ARRAY[0..32000] OF REAL;
	size : UINT;
END_VAR
VAR
	i: UINT;
	stop: UINT;
END_VAR

(*
version 1.5	16 mar 2008
programmer 	hugo
tested by		tobias

this function will calculate the median of a given array.
in order to do so the ariginal array is sorted and stays sorted after the function finishes
the function needs to be called:	_array_median(adr("array"),sizeof("array"));
this function will manipulate a given array.
the function will return the median of the original array.
for example [12,0,4,7,1] the median is 4 and the array after the function is called is [0,1,4,7,12]
because this function works with pointers its very time efficient and it needs no extra memory.

*)

_ARRAY_SORT(pt,size);
stop := SHR(size,2)-1;
IF EVEN(UINT_TO_INT(stop)) THEN
	_ARRAY_MEDIAN := pt^[SHR(stop,1)];
ELSE
	i := SHR(stop,1);
	_ARRAY_MEDIAN := (pt^[i] + pt^[i+1]) * 0.5;
END_IF;

(* old code
stop := (size - SIZEOF(pt)) / SIZEOF(pt);
FOR i := 0 TO stop - 1 DO
	FOR m := i + 1 TO stop DO
		IF pt^[i] > pt^[m] THEN
			temp := pt^[i];
			pt^[i] := pt^[m];
			pt^[m] := temp;
		END_IF;
	END_FOR;
END_FOR;
IF even(stop) THEN
	_array_median := pt^[stop/2];
ELSE
	i := stop/2;
	_array_median := (pt^[i] + pt^[i+1])/2;
END_IF;
*)
(* revision history
hm 	3.3.2007		rev 1.1
	corrected an error, changed the statement line 14	i := TRUNC(stop/2); to i := stop/2;

hm		22. sep 2007	rev 1.2
	changed algorithm to use _array_soft for performance reasons

hm		8. oct 2007		rev 1.3
	deleted unused variables m and temp

hm		14. nov 2007	rev 1.4
	corrected a problem with size calculation

hm		16.3. 2008		rev 1.5
	changed type of input size to uint
	performance improvements
*)

END_FUNCTION

// POUs/Mathematical/Array/_ARRAY_SORT
FUNCTION _ARRAY_SORT : BOOL
VAR_INPUT
	PT : POINTER TO ARRAY[1..32000] OF REAL;
	SIZE : UINT;
END_VAR
VAR
	stack_count: UINT;				(* Laufvariable Stack*)
	stack: ARRAY[1..32] OF UINT;	(* Stackgröße~ 1,6*Log(n)/log(2) *)
										(* Stackgröße 32 => ~1 Mio Elemente *)
	links: UINT;						(* Anfangselement des Arrays *)
	rechts: UINT;						(* Endelement des Arrays *)
	pivot: REAL;						(* temporärer Schwellwert für Tauschbedingung *)
	i: UINT;							(* Laufvariable1 *)
	j: UINT;							(* Laufvariable2 *)
	ende_innen: BOOL;				(* Ende innere Schleife *)
	ende_aussen: BOOL;				(* Ende äußere Schleife *)
	tmp: REAL;						(* Hilfsvariable zum Tauschen von Werten *)
END_VAR



(*
version 2.0	19. jan. 2011
programmer 	Alexander Trikitis
tested by	oscat

this function will sort a given array.
the function needs to be called:	_array_sort(adr("array"),sizeof("array"));
this function will manipulate a given array.
the function will not return anything except true, it will instead manipulate the original array.
because this function works with pointers its very time efficient and it needs no extra memory.

*)

(* Startwerte zur Arraygröße *)
links := 1;					(* Anfangselement des Arrays *)
rechts := SHR(size,2);		(* Endelement des Arrays *)
stack_count := 1;			(* Laufvariable Stack *)

WHILE NOT ende_aussen DO						(* äußere Schleife *)
	IF links < rechts THEN
		pivot := PT^[SHR(rechts+links,1)];			(* Wert des mittleren Elements als Pivot-Wert *)
		i := links -1;
		j := rechts +1;

		(* innere Schleife, teile Feld *)
		ende_innen := FALSE;
		REPEAT

			(* steigende Reihenfolge *)
			REPEAT	i := i+1;	UNTIL (PT^[i] >= pivot) OR NOT (i < rechts)	END_REPEAT;
			REPEAT	j := j-1;	UNTIL (PT^[j] <= pivot) OR NOT (j > links)	END_REPEAT;


			(*sinkende Reihenfolge *)
(*			REPEAT	i := i+1;	UNTIL (PT^[i] <= pivot) OR NOT (i < rechts)	END_REPEAT	*)
(*			REPEAT	j := j-1;	UNTIL (PT^[j] >= pivot) OR NOT (j > links)	END_REPEAT	*)

			IF i >= j THEN
				ende_innen := TRUE;
			ELSE
				   tmp := PT^[j];
				PT^[j] := PT^[i];
				PT^[i] := tmp;
			END_IF;

		UNTIL ende_innen END_REPEAT;

		(* Push stack *)
		stack[stack_count] := rechts;		(* rechten Teil später sortieren *)
		IF Stack_count < 32 THEN
			stack_count := stack_count +1;
		ELSE
			ende_aussen := TRUE;
			_ARRAY_SORT := FALSE;					(* Fehler: Stack zu klein *)
		END_IF;

		(* linken Teil sortiern *)
		rechts := MAX(links, i-1);

	ELSE

		IF stack_count = 1 THEN
			ende_aussen := TRUE;
		ELSE

			links := rechts+1;

			(* pop stack *)
			stack_count := stack_count -1;		(* jetzt rechten Teil sortierne *)
			rechts:= stack[stack_count];
		END_IF;

	END_IF;

END_WHILE;

_ARRAY_SORT := TRUE;				(* Sortierung beendet *)


(* algorithm used before rev 2.0

size := SHR(size,2);
size2 := UINT_TO_INT(SHR(size,1));
FOR i := SIZE2  TO 1 BY -1 DO
	j:=i;
    WHILE j <= SIZE2 DO
     	stop := j * 2 + 1;
        IF stop > UINT_TO_INT(SIZE) THEN stop := stop - 1;
        ELSIF pt^[stop-1] > pt^[stop] THEN stop := stop - 1;
		END_IF;
        IF pt^[j] < pt^[stop] THEN
         	temp := pt^[j];
            pt^[j] := pt^[stop];
            pt^[stop] := temp;
        END_IF;
        j := stop;
    END_WHILE;
END_FOR;

*)

(* heapsort
FOR heapsize := UINT_TO_INT(size) TO 1 BY -1 DO
	popmax := pt^[1];
	pt^[1] := pt^[heapsize];
   	i := 1;
	hs2 := SHR(heapsize,1);
	WHILE i <= hs2 DO
       	stop := i * 2 + 1;  
        	IF stop > heapsize THEN stop := stop - 1;
        	ELSIF pt^[stop-1] > pt^[stop] THEN stop := stop - 1;
	 	END_IF;
        	IF pt^[i] < pt^[stop] THEN
            		temp := pt^[i];
            		pt^[i] := pt^[stop];
            		pt^[stop] := temp;
        	END_IF;
        	i := stop;
    	END_WHILE;
	pt^[heapsize] := popmax;
END_FOR;

_ARRAY_SORT2 := TRUE;
*)

(* old algorithm bubble sort used before rev 1.2
stop := (size - SIZEOF(pt)) / SIZEOF(pt);
FOR i := 0 TO stop - 1 DO
	FOR m := i + 1 TO stop DO
		IF pt^[i] > pt^[m] THEN
			temp := pt^[i];
			pt^[i] := pt^[m];
			pt^[m] := temp;
		END_IF;
	END_FOR;
END_FOR;
_array_sort := TRUE;

*)


(* revision history

hm 	6.1.2007 	rev 1.1
	changed return value to true

hm	22. sep 2007	rev 1.2
	changed sorting algorithm to heap sort for performance reasons

hm 	14. nov 2007	rev 1.3
	changed calculation of stop to be more efficient

hm	15 dec 2007	rev 1.4
	added function return true

hm	5. jan 2008		rev 1.5
	improved performance

hm	16. mar. 2008	rev 1.6
	changed type of input size to uint

hm	28. mar. 2008	rev 1.7
	changed input f to pt

hm	19. jan. 2011	rev 2.0
	new faster algorithm using qucksort (Alexander Drikitis)

*)

END_FUNCTION

// POUs/Mathematical/EVEN
FUNCTION EVEN : BOOL
VAR_INPUT
	in : DINT;
END_VAR


(*
version 1.1	1 dec 2007
programmer 	hugo
tested by		tobias

this function chacks an input for even  value
the output is true if the input is even.
execution time on wago 750 - 841 =  10  us
*)

EVEN := NOT in.0;

(* revision history
hm	1. oct 2006	rev 1.0
	ORIGINAL VERSION

hm	01.12.2007	rev 1.1
	changed code for improved performance

hm	21. mar. 2008	rev 1.2
	changed type of input IN from INT to DINT
*)

END_FUNCTION

// POUs/Mathematical/Array/_ARRAY_MUL
FUNCTION _ARRAY_MUL : BOOL
VAR_INPUT
	pt : POINTER TO ARRAY[0..32000] OF REAL;
	size : UINT;
	X : REAL;
END_VAR
VAR
	i: UINT;
	stop: UINT;
END_VAR

(*
version 1.0	2. apr. 2008
programmer 	hugo
tested by	tobias

this function will multiply each element of the array and stroe the result instead of the element.
Array[i] := ARRAY[i] * X.
the function needs to be called:	array_avg(adr("array"),sizeof("array"));
because this function works with pointers its very time efficient and it needs no extra memory.

*)

stop := SHR(size,2)-1;
FOR i := 0 TO stop DO
	PT^[i] := PT^[i] * X;
END_FOR;
_ARRAY_MUL := TRUE;


(* revision history
hm	2. apr 2008		rev 1.0
	original version

*)

END_FUNCTION

// POUs/Mathematical/Array/_ARRAY_SHUFFLE
FUNCTION _ARRAY_SHUFFLE : BOOL
VAR_INPUT
	pt : POINTER TO ARRAY[0..32000] OF REAL;
	size : UINT;
END_VAR
VAR
	temp : REAL;
	pos  : INT;
	i: INT;
	stop: INT;
END_VAR


(*
version 1.2	30. mar. 2008
programmer 	kurt
tested by		hugo

this function will randomly shuffle the elements of an array
*)

stop := UINT_TO_INT(SHR(size,2)-1);
FOR i := 0 TO stop DO
        pos := RDM2(i+pos,0,stop);
        (* swap elements *)
        temp := pt^[i];
        pt^[i] := pt^[pos];
        pt^[pos] := temp;
END_FOR;

_ARRAY_SHUFFLE := TRUE;


(* revision History
hm 	4. mar 2008	rev 1.0
	original version

hm	16. mar. 2008	rev 1.1
	changed type of input size to uint

hm	30. mar. 2008	rev 1.2
	changed last in rdm2 fromm pos to i + pos to allow for more randomness

*)

END_FUNCTION

// POUs/Mathematical/RDM2
FUNCTION RDM2 : INT
VAR_INPUT
	last : INT;
	low : INT;
	high : INT;
END_VAR


(*
version 1.1	18. oct. 2008
programmer 	hugo
tested by	tobias

this function calculates an integer pseudo random number
the random number will be in the range of low <= rdm2 <= high.

*)

RDM2 := TRUNC_INT(RDM(FRACT(last * math.PI)) * (high - low + 1)) + low;

(* revision history
hm		29. feb 2008		rev 1.0
	original version

hm		18. oct. 2008		rev 1.1
	using math constants

*)

END_FUNCTION

// POUs/Mathematical/RDM
FUNCTION RDM : REAL
VAR_INPUT
	last : REAL;
END_VAR
VAR
	tn : DWORD;
	tc : INT;
END_VAR


(*
version 1.9	10. mar. 2009
programmer 	hugo
tested by		tobias

this function calculates a pseudo random number
to generate the number it reads the sps timer and calculates a random number between 0 and 1:
in order to use rdm more then once within one sps cycle it need to be called with different seed numbers LAST.

*)

tn := T_PLC_MS();
tc := BIT_COUNT(tn);
tn.31 := tn.2;
tn.30 := tn.5;
tn.29 := tn.4;
tn.28 := tn.1;
tn.27 := tn.0;
tn.26 := tn.7;
tn.25 := tn.6;
tn.24 := tn.3;
tn := ROL(tn,BIT_COUNT(tn)) OR 16#80000001;
tn := tn MOD 71474513 + INT_TO_DWORD(tc + 77);
RDM := FRACT(DWORD_TO_REAL(tn) / 10000000.0 * (math.E - LIMIT(0.0,last,1.0)));


(*
pt := ADR(temp);
pt^ := (T_PLC_MS() AND 16#007FFFFF) OR 16#3D000000;
RDM := fract(modR(temp*e+pi1, PI1-last) + modR(temp*PI1+e + last,e-last));
*)

(* revision history
hm		16. jan 2007		rev 1.0
	original version

hm		11. nov 2007		rev 1.1
	changed time() into t_plc_ms()

hm		20. nov 2007		rev 1.2
	changed code of temp calculation to avoid overflow in modr due to resuclt would not fit DINT for high timeer values

hm		5. jan 2008		rev 1.3
	changed calculation of temp to avoid problem with high values of t_plc_ms

hm		2. feb 2008		rev 1.4
	changed algorithm to avoind non iec functions and guarantee more randomness

hm	10. mar. 2008		rev 1.5
	make sure last will be between 0 and 1 to avoid invalid results

hm	16. mar. 2008		rev 1.6
	added conversion for tc to avoid warnings under codesys 3.0

hm	18. may. 2008		rev 1.7
	changed constant E to E1

hm	18. oct. 2008		rev 1.8
	using math constants

hm	10. mar. 2009		rev 1.9
	real constants updated to new systax using dot

*)

END_FUNCTION

// POUs/Logic/gate logic/BIT_COUNT
FUNCTION BIT_COUNT : INT
VAR_INPUT
	IN : DWORD;
END_VAR


(*
version 1.1	10 sep 2007
programmer 	hugo
tested by		tobias

BIT_COUNT counts the amount True of bits in a dword.
for exabple: bit_count(3) returns 2 because two bits (bits 0 and 1) are true and all others are false. 

*)

WHILE in > 0 DO
	IF in.0 THEN Bit_Count := Bit_Count + 1; END_IF;
	in := SHR(in,1);
END_WHILE;



(* revision history
5.7.2007	rev 1.0		original version

10.9.2007	rev 1.1		hm
	changed algorithm for better performace
	the execution time has reduced by a factor of 5
	deleted unused variable temp
*)

END_FUNCTION

// POUs/Mathematical/FRACT
FUNCTION FRACT : REAL
VAR_INPUT
	x : REAL;
END_VAR


(*
version 1.3	10. mar. 2009
programmer 	hugo
tested by		tobias

this function returns the fraction of a real number
fract(3.14) = 0.14

*)

IF ABS(x) < 2.0E9 THEN
	FRACT := x - DINT_TO_REAL(D_TRUNC(x));
ELSE
	FRACT := 0.0;
END_IF;

(* revision history
hm	4. aug 2006	rev 1.0
	original version

hm	11. mar 2008	rev 1.1
	added dint_to_real for compatibility reasons
	now returns 0 for number > 2e9
	changed input to x

hm	21. mar. 2008	rev 1.2
	use D_trunc instead of TRUNC for compatibility reasons

hm	10. mar. 2009	rev 1.3
	real constants updated to new systax using dot

*)

END_FUNCTION

// POUs/Mathematical/D_TRUNC
FUNCTION D_TRUNC : DINT
VAR_INPUT
	X : REAL;
END_VAR

(*
version 1.2	10. mar. 2009
programmer 	hugo
tested by		oscat

d_trunc truncates a real to a dint 1.5 will be 1 and -1.5 will be -1
d_trunc is necessary because many systems do not offer a trunc to a dint
also real_to_dint will not deliver the same result on different systems

*)

D_TRUNC := REAL_TO_DINT(X);
IF X > 0.0 THEN
	IF DINT_TO_REAL(D_TRUNC) > X THEN D_TRUNC := D_TRUNC - 1; END_IF;
ELSE
	IF DINT_TO_REAL(D_TRUNC) < X THEN D_TRUNC := D_TRUNC + 1; END_IF;
END_IF;


(* for systems that support a dint truncation this routine can be replaced by trunc() *)


(* revision history
hm	21. mar. 2008	rev 1.0
	original version

hm	31. oct. 2008	rev 1.1
	optimized performance

hm	10. mar. 2009	rev 1.2
	real constants updated to new systax using dot
*)

END_FUNCTION

// POUs/Mathematical/MODR
FUNCTION MODR : REAL
VAR_INPUT
	IN : REAL;
	DIVI : REAL;
END_VAR


(*
version 1.5	10. mar. 2009
programmer 	hugo
tested by		tobias

this is a modulo funtion for real numbers
modr(5.5,2.5) = 0.5

*)

IF divi = 0.0 THEN
	MODR := 0.0;
ELSE
	MODR := in - DINT_TO_REAL(FLOOR2(in / divi)) * divi;
END_IF;

(* revision history

hm	4. aug.2006		rev 1.0

hm	28. jan.2007	rev 1.1
	modr(x,0) will deliver the result 0

hm	21. mar 2008	rev 1.2
	use D_trunc for compatibility reasons

hm	4. apr. 2008	rev 1.3
	added type conversion to avoid warnings under codesys 3.0

hm	31. oct. 2008	rev 1.4
	changed algorithm to the more common version using floor instead of TRUNC

hm	10. mar. 2009	rev 1.5
	real constants updated to new systax using dot

*)

END_FUNCTION

// POUs/Mathematical/FLOOR2
FUNCTION FLOOR2 : DINT
VAR_INPUT
	X : REAL;
END_VAR



(*
version 1.1	4. apr. 2008
programmer 	hugo
tested by		tobias

This is a rounding function which returns the biggest possible integer which is less or equal to X.
floor2(3.14) = 3
floor2(-3.14) = -4

*)

FLOOR2 := REAL_TO_DINT(X);
IF DINT_TO_REAL(FLOOR2) > X THEN
	FLOOR2 := FLOOR2 - 1;
END_IF;

(* revision history
hm	21. mar. 2008	rev 1.0
	originlal version

hm	4. apr. 2008	rev 1.1
	added type conversion to avoid warnings under codesys 3.0
*)

END_FUNCTION

// POUs/Mathematical/FLOOR
FUNCTION FLOOR : INT
VAR_INPUT
	X : REAL;
END_VAR


(*
version 1.1	21. mar. 2008
programmer 	hugo
tested by		tobias

This is a rounding function which returns the biggest possible integer which is less or equal to X.
floor(3.14) = 3
floor(-3.14) = -4

*)

FLOOR := REAL_TO_INT(X);
IF FLOOR > X THEN
	FLOOR := FLOOR - 1;
END_IF;

(* revision history
hm		7. feb 2007		rev 1.0
	originlal version

hm		21. mar. 2008	rev 1.1
	replaced trunc with real_to_int for compatibility reasons

*)

END_FUNCTION

// POUs/Buffer Management/_BUFFER_CLEAR
FUNCTION _BUFFER_CLEAR : BOOL
VAR_INPUT
	PT : POINTER TO BYTE;
	SIZE : UINT;
END_VAR
VAR
	ptw : POINTER TO DWORD;
	temp: DWORD;
	end, end32 : DWORD;
END_VAR


(*
version 1.2	31. oct. 2008
programmer 	hugo
tested by	oscat

this function will initialize a given array of byte with 0.
the function needs to be called:	_buffer_clear(adr("array"),sizeof("array"));
this function will manipulate a given array.
the function manipulates the original array, it rerturnes true when finished.
because this function works with pointers its very time efficient and it needs no extra memory.

*)

(* this routine uses 32 bit access to gain speed *)
(* first access bytes till pointer is aligned for 32 bit access *)
temp := pt;
end := temp + UINT_TO_DWORD(size);
end32 := end - 3;
WHILE (pt < end) AND ((temp AND 16#00000003) > 0) DO
	pt^ := 0;
	pt := pt + 1;
	temp := temp + 1;
END_WHILE;
(* pointer is aligned, now copy 32 bits at a time *)
ptw := pt;
WHILE ptw < end32 DO (* *)
	ptw^ := 0;
	ptw := ptw + 4;
END_WHILE;
(* copy the remaining bytes in byte mode *)
pt := ptw;
WHILE pt < end DO
	pt^ := 0;
	pt := pt + 1;
END_WHILE;

_BUFFER_CLEAR := TRUE;

(* revision History
hm 	5. mar. 2008	rev 1.0
	original version

hm	16. mar. 2008	rev 1.1
	added type conversion to avoid warnings under codesys 30
	chaged type of input size to uint
	deleted unused variable i

hm	31. oct. 2008	rev 1.2
	corrected an error while routine would write outside of arrays

*)

END_FUNCTION

// POUs/Buffer Management/_BUFFER_INIT
FUNCTION _BUFFER_INIT : BOOL
VAR_INPUT
	PT : POINTER TO BYTE;
	SIZE : UINT;
	INIT : BYTE;
END_VAR
VAR
	ptw : POINTER TO DWORD;
	temp : DWORD;
	end, end32 : DWORD;
END_VAR


(*
version 1.2	31. oct. 2008
programmer 	hugo
tested by	oscat

this function will initialize a given array of byte with init.
the function needs to be called:	_buffer_init(adr("array"),sizeof("array"),init);
this function will manipulate a given array.
the function manipulates the original array, it rerturnes true when finished.
because this function works with pointers its very time efficient and it needs no extra memory.

*)

(* this routine uses 32 bit access to gain speed *)
(* first access bytes till pointer is aligned for 32 bit access *)
temp := pt;
end := temp + UINT_TO_DWORD(size);
end32 := end - 3;
WHILE (pt < end) AND ((temp AND 16#00000003) > 0) DO
	pt^ := init;
	pt := pt + 1;
	temp := temp + 1;
END_WHILE;
(* pointer is aligned, now copy 32 bits at a time *)
ptw := pt;
temp := SHL(BYTE_TO_DWORD(init),24) OR SHL(BYTE_TO_DWORD(init),16) OR SHL(BYTE_TO_DWORD(init),8) OR BYTE_TO_DWORD(init);
WHILE ptw < end32 DO
	ptw^ := temp;
	ptw := ptw + 4;
END_WHILE;
(* copy the remaining bytes in byte mode *)
pt := ptw;
WHILE pt < end DO
	pt^ := init;
	pt := pt + 1;
END_WHILE;

_BUFFER_INIT := TRUE;

(* revision History
hm 	5. mar. 2008	rev 1.0
	original version

hm	16. mar. 2008	rev 1.1
	added type conversion to avoid warnings under codesys 3.0
	chaged type of input size to uint.

hm	31. oct. 2008	rev 1.2
	corrected an error while routine would write outside of arrays

*)

END_FUNCTION

// POUs/Buffer Management/_BUFFER_INSERT
FUNCTION _BUFFER_INSERT : INT
VAR_INPUT
	STR : STRING(STRING_LENGTH);
	POS : INT;
	PT : POINTER TO ARRAY[0..32767] OF BYTE;
	SIZE : UINT;
END_VAR
VAR
	end : INT;
	lx: INT;
	i: INT;
END_VAR


(*
version 1.5	2. jan. 2012
programmer 	hugo
tested by	oscat

this function will insert a string at a given position in a buffer.
the function needs to be called:	_buffer_init(adr("array"),sizeof("array"),init);
this function will manipulate a given array.
the function manipulates the original array, it returnes the next position after the input string when finished.
because this function works with pointers its very time efficient and it needs no extra memory.

*)

lx := LEN(str);
end := pos + lx;
(* first move the upper part of the buffer to make space for the string *)
FOR i := UINT_TO_INT(size) - 1 TO end BY -1 DO
	pt^[i] := pt^[i-lx];
END_FOR;
(* copy the string *)
_BUFFER_INSERT := _STRING_TO_BUFFER(str, pos, PT, size);


(* revision History
hm 	9. mar. 2008	rev 1.0
	original version

hm	16. mar. 2008	rev 1.1
	changed type of input size to uint

hm	13. may. 2008	rev 1.2
	changed type of pointer to array[1..32767]
	changed size of string to STRING_LENGTH

hm	23. mar. 2009	rev 1.3
	avoid writing to input pos

hm	12. nov. 2009	rev 1.4
	code optimized

hm 2. jan 2012	rev 1.5
	function now returns the next position after the input string

*)

END_FUNCTION

// POUs/Buffer Management/_STRING_TO_BUFFER
FUNCTION _STRING_TO_BUFFER : INT
VAR_INPUT
	STR : STRING(STRING_LENGTH);
	POS : INT;
	PT : POINTER TO ARRAY[0..32767] OF BYTE;
	SIZE : UINT;
END_VAR
VAR
	ps : POINTER TO BYTE;
	i: INT;
	end: INT;
END_VAR


(*
version 1.4	2. jan. 2012
programmer 	hugo
tested by		oscat

this function will copy a string into an array of byte starting at position pos.
the function needs to be called:	_String_To_buffer(str, pos, adr("array"),sizeof("array"));
this function will manipulate the array directly in memory and returns the position after the input string when finished.
because this function works with pointers its very time efficient and it needs no extra memory.

*)

ps := ADR(str);
end := MIN(pos + LEN(str), UINT_TO_INT(size));
IF end > 0 THEN end := end -1; END_IF;
FOR i := pos TO end DO
	pt^[i] := ps^;
	ps := ps + 1;
END_FOR;

_STRING_TO_BUFFER := i;

(* revision History

hm 	5. mar. 2008	rev 1.0
	original version

hm	16. mar. 2008	rev 1.1
	changed type of input size to uint

hm	13. may. 2008	rev 1.2
	changed type of pointer to array[1..32767]
	changed size of string to STRING_LENGTH

hm	12. nov. 2009	rev 1.3
	limit end to size - 1

hm	2. jan 2012	rev 1.4
	return the position after the input string when finished
*)

END_FUNCTION

// POUs/Buffer Management/_BUFFER_UPPERCASE
FUNCTION _BUFFER_UPPERCASE : BOOL
VAR_INPUT
	PT : POINTER TO ARRAY[0..32000] OF BYTE;
	SIZE : INT;
END_VAR
VAR
	pos: INT;
END_VAR


(*
version 1.0	20. jan. 2011
programmer 	hugo
tested by	oscat

this function will convert an array of byte into uppercase
the function needs to be called:	_buffer_clear(adr("array"),sizeof("array"));
this function will manipulate a given array.
the function manipulates the original array, it rerturnes true when finished.
because this function works with pointers its very time efficient and it needs no extra memory.

*)

pos := 0;
WHILE pos < size DO
	PT^[pos] := TO_UPPER(pt^[pos]);
	pos := pos + 1;
END_WHILE;

_BUFFER_UPPERCASE := TRUE;

(* revision History
hm 	20. jan. 2011	rev 1.0
	original version

*)

END_FUNCTION

// POUs/String/TO_UPPER
FUNCTION TO_UPPER : BYTE
VAR_INPUT
	IN : BYTE;
END_VAR


(*
version 1.3	16. jan. 2009
programmer 	hugo
tested by		oscat

to_upper converts a character from lowercase to uppercase

*)

IF in > 96 AND in < 123 THEN
   TO_UPPER := in AND 16#DF;
ELSIF in > 223 AND in <> 247 AND in <> 255 AND setup.EXTENDED_ASCII THEN
   TO_UPPER := in AND 16#DF;
ELSE
   TO_UPPER := in;
END_IF;




(* revision history
hm	6. mar. 2008	rev 1.0
	original version

hm	19. oct. 2008	rev 1.1
	changed setup constants

ks	25. oct. 2008	rev 1.2
	optimized code

hm 16. jan 2009	rev 1.3
	corrected an error in module

*)

END_FUNCTION

// POUs/String/LOWERCASE
FUNCTION LOWERCASE : STRING(STRING_LENGTH)
VAR_INPUT
	str : STRING(STRING_LENGTH);
END_VAR
VAR
	PT : POINTER TO BYTE;
	pos: INT;
	l: INT;
END_VAR

(*
version 1.3	29. mar. 2008
programmer 	hugo
tested by		tobias

lowercase returns str while all letters A..Z and Ä.Ö,Ü are converted to lowercase.

*)

PT := ADR(LOWERCASE);
lowercase := str;
l := LEN(str);
FOR pos := 1 TO l DO
	pt^ := TO_LOWER(pt^);
	PT := PT + 1;
END_FOR;

(* revision histroy
hm	6. oct. 2006	rev 1.0
	original release

hm	4. feb. 2008	rev 1.1
	improved performance
	added Ä.Ö,Ü

hm	6. mar. 2008	rev 1.2
	added support for exteded Ascii

hm	29. mar. 2008	rev 1.3
	changed STRING to STRING(STRING_LENGTH)
*)

END_FUNCTION

// POUs/String/TO_LOWER
FUNCTION TO_LOWER : BYTE
VAR_INPUT
	IN : BYTE;
END_VAR


(*
version 1.2	25. oct 2008
programmer 	hugo
tested by		tobias

to_lower converts a character from uppercase to lowercase

*)

IF in > 64 AND in < 91 THEN
   TO_LOWER := in OR 16#20;
ELSIF (in > 191 AND in < 223) AND in <> 215 AND setup.EXTENDED_ASCII THEN
   TO_LOWER := in OR 16#20;
ELSE
   TO_LOWER := in;
END_IF;


(* revision history
hm	6. mar. 2008	rev 1.0
	original version

hm	19. oct. 2008	rev 1.1
	changed setup constants

ks	25. oct. 2008	rev 1.2
	optimized code
*)

END_FUNCTION

// POUs/String/UPPERCASE
FUNCTION UPPERCASE : STRING(STRING_LENGTH)
VAR_INPUT
	str : STRING(STRING_LENGTH);
END_VAR
VAR
	pt : POINTER TO BYTE;
	pos: INT;
	l: INT;
END_VAR

(*
version 1.3	29. mar. 2008
programmer 	hugo
tested by	tobias

uppercase returns str while all letters a..z and ä,ö,ü are converted to uppercase

*)

pt := ADR(UPPERCASE);
UPPERCASE := str;
l := LEN(str);
FOR pos := 1 TO l DO
	pt^ := TO_UPPER(pt^);
	pt := pt + 1;
END_FOR;

(* revision histroy
hm	6. oct. 2006	rev 1.0
	original release

hm	4. feb. 2008	rev 1.1
	improved performance
	added Ä,Ö,Ü

hm	6. mar. 2008	rev 1.2
	added support for exteded Ascii

hm	29. mar. 2008	rev 1.3
	changed STRING to STRING(STRING_LENGTH)

*)

END_FUNCTION

// POUs/Engineering/signal generators/_RMP_B
FUNCTION_BLOCK _RMP_B
VAR_INPUT
	DIR : BOOL;  (* true = up *)
	E : BOOL := TRUE;
	TR : TIME;
END_VAR
VAR_IN_OUT
	RMP : BYTE;
END_VAR
VAR
	tx, tl, tn : TIME;
	init : BOOL;
	last_dir : BOOL;
	start : BYTE;
END_VAR


(*
version 1.2		19. feb. 2011
programmer 	hugo
tested by		oscat

_RMP_B generates a ramp on an external var of type byte
tr is the total ramp time, E is an enable and dir the direction of the ramp

*)

(* read system timer *)
tx := DWORD_TO_TIME(T_PLC_MS());

IF E AND init AND (dir = last_dir) AND (RMP <> SEL(DIR, 0, 255)) AND TR = tn THEN
	RMP := FRMP_B(start, DIR, tx - tl, TR);
ELSE
	init := TRUE;
	tl := tx;
	tn := tr;
	start := RMP;
END_IF;
last_dir := dir;



(* revison history
hm	22. oct. 2008	rev 1.0
	original version

hm	20. nov. 2008	rev 1.1
	set default for E to be TRUE
	added init

hm	19. nov. 2011	rev 1.2
	new code
*)

END_FUNCTION_BLOCK

// POUs/Mathematical/functions/FRMP_B
FUNCTION FRMP_B : BYTE
VAR_INPUT
	START : BYTE;
	DIR : BOOL;
	TD : TIME;
	TR : TIME;
END_VAR
VAR
END_VAR


(*
version 1.0		17. feb. 2011
programmer 	hugo
tested by		oscat

this function calculates a ramp and limits the output to 0 .. 255 without overflow problems

*)

IF TD < TR THEN
	FRMP_B := MIN(DWORD_TO_BYTE(SHL(TIME_TO_DWORD(TD), 8) / TIME_TO_DWORD(TR)), SEL(DIR, START, BYTE#255 - START));
	IF DIR THEN
		FRMP_B := START + FRMP_B;
	ELSE
		FRMP_B := START - FRMP_B;
	END_IF;
ELSE
	FRMP_B := SEL(DIR, 0, 255);
END_IF;


(* revision history

17. feb. 2011	rev 1.0
	new module

*)

END_FUNCTION

// POUs/Engineering/signal generators/_RMP_NEXT
FUNCTION_BLOCK _RMP_NEXT
VAR_INPUT
	E : BOOL := TRUE;
	IN : BYTE;
	TR : TIME;
	TF : TIME;
	TL : TIME;
END_VAR
VAR_OUTPUT
	DIR : BOOL;    (* upwards = TRUE *)
	UP : BOOL;
	DN : BOOL;
END_VAR
VAR_IN_OUT
	OUT : BYTE;
END_VAR
VAR
	rmx : _RMP_B;
	dirx : TREND_DW;
	t_lock :TP;
	xen: BOOL;
	xdir: BOOL;
END_VAR


(*
version 1.4		18. jul. 2009
programmer 	hugo
tested by		oscat


_RMP_NEXT  will generate a ramp output following the input IN.
on a rising ramp the output will stop as soon as it has surpassed the input in, and on a falling ramp it will stop when out is smaller than in.
a lockout time T_L will be added between up and down direction.

*)

dirx(X := in);

t_lock(in := FALSE, pt := TL);

IF dirx.TU AND (OUT < IN) THEN
	IF NOT xdir AND xen THEN t_lock(in := TRUE); END_IF;
	xen := TRUE;
	xdir := TRUE;
ELSIF dirx.TD AND (OUT > IN) THEN
	IF xdir AND xen THEN t_lock(in := TRUE); END_IF;
	xen := TRUE;
	xdir := FALSE;
ELSIF xen THEN
	IF (xdir AND (out >= in)) OR (NOT xdir AND (out <= in)) THEN
		xen := FALSE;
		IF tl > t#0s THEN t_lock(IN := TRUE); END_IF;
	END_IF;
END_IF;

IF NOT t_lock.Q AND xen THEN
		UP := XDIR;
		DIR := XDIR;
		DN := NOT XDIR;
ELSE
	UP := FALSE;
	DN := FALSE;
END_IF;

rmx(rmp := OUT, E := E AND (UP OR DN) , dir := DIR, tr := SEL(dir, TF, TR));


(* revison history
hm	23. nov. 2008	rev 1.0
	original version

hm	24. jan. 2009	rev 1.1
	deleted unused vars tmp1, tmp2

hm	20. feb. 2009	rev 1.2
	improved algorithm
	added TL

hm	9. mar. 2009	rev 1.3
	input E was ignored
	removed double assignments

hm	18. jul. 2009	rev 1.4
	improved performance

*)

END_FUNCTION_BLOCK

// POUs/Engineering/signal processing/TREND_DW
FUNCTION_BLOCK TREND_DW
VAR_INPUT
	X : DWORD;
END_VAR
VAR_OUTPUT
	Q : BOOL;
	TU : BOOL;
	TD : BOOL;
	D : DWORD;
END_VAR
VAR
	last_X: DWORD;
END_VAR

(*
version 1.2	14. mar. 2009
programmer 	hugo
tested by		oscat

trend_DW analyses the trend of a input signal.
The Output Q is True if the input X is >= last_X and is false if the input X is <= last_X
in addition to the trend the output TU will be high for one cycle to signal a rising of the input value X
and  TD will signal a decreasing value on the input X.
in case of a change the output D will show the delta of the input to the last input value.


*)

IF X > last_X THEN
	TU := TRUE;
	TD := FALSE;
	D := X - last_X;
	Q := TRUE;
ELSIF X < last_X THEN
	TD := TRUE;
	TU := FALSE;
	D := last_X - X;
	Q := FALSE;
ELSE
	TU := FALSE;
	TD := FALSE;
	D := 0;
END_IF;
last_X := X;



(* revision history
hm	21. nov. 2008	rev 1.0
	original version

hm	20. feb. 2009	rev 1.1
	added outputs TU, TD and D

hm	14. mar. 2009	rev 1.2
	removed double assignments

*)

END_FUNCTION_BLOCK

// POUs/Engineering/signal processing/TREND
FUNCTION_BLOCK TREND
VAR_INPUT
	X : REAL;
END_VAR
VAR_OUTPUT
	Q : BOOL;
	TU : BOOL;
	TD : BOOL;
	D : REAL;
END_VAR
VAR
	last_X: REAL;
END_VAR

(*
version 1.0	21. aug. 2009
programmer 	hugo
tested by		oscat

trend analyses the trend of a input signal.
The Output Q is True if the input X is >= last_X and is false if the input X is <= last_X
in addition to the trend the output TU will be high for one cycle to signal a rising of the input value X
and  TD will signal a decreasing value on the input X.
in case of a change the output D will show the delta of the input to the last input value.

*)

TU := X > last_X;
TD := X < last_X;
Q := TU OR TD;
D := X - LAST_X;

last_X := X;



(* revision history
hm	21. aug. 2009	rev 1.0
	original version

*)

END_FUNCTION_BLOCK

// POUs/Engineering/signal generators/_RMP_W
FUNCTION_BLOCK _RMP_W
VAR_INPUT
	DIR : BOOL;
	E : BOOL := TRUE;
	TR : TIME;
END_VAR
VAR_IN_OUT
	RMP : WORD;
END_VAR
VAR
	tx, tl : DWORD;
	step : DINT;
	init: BOOL;
	last_dir : BOOL;
END_VAR


(*
version 1.1	20. nov. 2008
programmer 	hugo
tested by	oscat


_RMP_B generates a ramp on an external var of type byte
tr is the total ramp time, E is an enable and dir the direction of the ramp

*)

tx := T_PLC_MS();
IF E AND init THEN
	(* we need to set tl = tx when direction changes *)
	IF dir XOR last_dir THEN
	 tl := tx;
	 last_dir := dir;
	END_IF;
	(* check_elapsed time and calculate only if necessary *)
	IF tr > t#0s THEN
		step := DWORD_TO_DINT(SHL(tx-tl, 16) / TIME_TO_DWORD(TR));
	ELSE
		step := 65535;
	END_IF;
	IF step > 0 THEN
		(* perform the step on the ramp *)
		tl := tx;
		(* calculate the step response *)
		IF NOT dir THEN step := - step; END_IF;
		rmp := DINT_TO_WORD(LIMIT(0, WORD_TO_DINT(rmp) + step, 65535));
	END_IF;
ELSE
	tl := tx;
	init := TRUE;
END_IF;


(* revison history
hm	22. oct. 2008	rev 1.0
	original version

hm	20. nov. 2008	rev 1.1
	set default for E to be TRUE
	added init

*)

END_FUNCTION_BLOCK

// POUs/Logic/generators/A_TRIG
FUNCTION_BLOCK A_TRIG
VAR_INPUT
	IN : REAL;
	RES : REAL;
END_VAR
VAR_OUTPUT
	Q : BOOL;
	D : REAL;
END_VAR
VAR
	last_in : REAL;
END_VAR

(*
version 1.1	25. oct. 2008
programmer 	hugo
tested by	oscat

this block is similar to the IEC Standard R_trig and F_trig but it monitors a REAL for change.
if the valiue on IN changes more then D from the last value it will generate trigger and display the difference in output D.
the trigger will only be active for one cycle.

*)

D := IN - LAST_IN;
Q := ABS(D) > res;
IF Q THEN last_in := IN; END_IF;
D := IN - LAST_IN;


(* revision history

hm 	16. jul. 2008	rev 1.0
	original version released

hm	25. oct. 2008	rev 1.1
	code optimization
	a_trig now also works for res = 0

*)

END_FUNCTION_BLOCK

// POUs/Mathematical/ACOSH
FUNCTION ACOSH : REAL
VAR_INPUT
	X : REAL;
END_VAR


(*
version 1.3	10. mar. 2009
programmer 	hugo
tested by		tobias

this function calculates the arcus cos hyperbolicus

*)

ACOSH := LN(SQRT(X * X - 1.0) + X);

(* revision history
hm		12 jan 2007	rev 1.0
	original version

hm		2. dec 2007	rev 1.1
	changed code for better performance

hm	16. mar. 2007		rev 1.2
	changed sequence of calculations to improve performance

hm	10. mar. 2009		rev 1.3
	real constants updated to new systax using dot

*)

END_FUNCTION

// POUs/Mathematical/ACOTH
FUNCTION ACOTH : REAL
VAR_INPUT
	X : REAL;
END_VAR


(*
version 1.2	10. mar. 2009
programmer 	hugo
tested by		tobias

this function calculates the arcus cotangens hyperbolicus

*)

ACOTH := LN((x+1.0)/(x-1.0))*0.5;

(* revision history
hm		12 jan 2007	rev 1.0
	original version

hm		5. jan 2008	rev 1.1
	improved code for better performance

hm	10. mar. 2009		rev 1.2
	real constants updated to new systax using dot

*)

END_FUNCTION

// POUs/Mathematical/AGDF
FUNCTION AGDF : REAL
VAR_INPUT
	X : REAL;
END_VAR


(*
version 1.1	10. mar. 2009
programmer 	hugo
tested by		tobias

this function calculates the inverse Gudermannian function.

*)

AGDF := LN((1.0 + SIN(X)) / COS(X));

(* comment
the current implementation gives sufficient accuracy only up to X = 1.57 or an output > 10.
is X closer to PI/2 then the function is more and more unreliable
*)



(* revision history
hm	27. apr. 2008	rev 1.0
	original version

hm	10. mar. 2009	rev 1.1
	real constants updated to new systax using dot

*)

END_FUNCTION

// POUs/Engineering/signal processing/AIN
FUNCTION AIN : REAL
VAR_INPUT
	in : DWORD;
END_VAR
VAR_INPUT CONSTANT
	Bits : BYTE;
	sign : BYTE := 255;
	low : REAL;
	high : REAL := 10.0;
END_VAR
VAR CONSTANT
	ff : DWORD := 16#FFFFFFFF;
END_VAR
VAR
	temp1 : DWORD;
	temp2 : DWORD;
	sx : BOOL;
END_VAR

(*
version 1.5	16 mar 2008
programmer 	oscat
tested by		tobias

Ain converts signals from A/D converters or other digital sources to an internal real value
the lowest number of bits are extracted from the input word and the sign will be extracted if available separately.
the output signal is then conditioned to range from low to high values for a 0 to max value on the analog inputs:
for example a 15bit input (bits := 12) with sign at bit 15 (0..15) will deliver 0.0 (low value at 0) for an input value of 2#0000_0000_0000
an input value of 2#1111_1111_1111 will deliver 10.0 on the output (high value set to 10).

*)

(* extract the sign bit *)
IF sign < 32 THEN
	temp1 := SHR(in,sign);
	sx := temp1.0;
ELSE
	sx := FALSE;
END_IF;
temp1 := SHR(ff, 32-bits);
temp2 := in AND temp1;
AIN := (high - low) * DWORD_TO_REAL(temp2) / DWORD_TO_REAL(temp1) + low;
IF sx THEN AIN := -AIN; END_IF;

(* revision history
hm 18.8.2006	rev 1.1
	fixed an error with low value negative and high value 0.

hm 19.1.2007	rev 1.2
	fixed an error with sign bit.

hm	13.9.2007	rev 1.3
	changed code to avoid warning under codesys 2.8.1

hm	2. dec 2007	rev 1.4
	changed code for better performance

hm	16. mar 2008	rev 1.5
	added type conversions to avoid warnings under codesys 30
*)

END_FUNCTION

// POUs/Engineering/signal processing/AIN1
FUNCTION_BLOCK AIN1
VAR_INPUT
	in : DWORD;
END_VAR
VAR_INPUT CONSTANT
	sign_bit : INT := 255;
	error_bit : INT := 255;
	error_code_en : BOOL;
	error_code : DWORD;
	overflow_bit : INT := 255;
	overflow_code_en : BOOL;
	overflow_code : DWORD;
	Bit_0 : INT;
	Bit_N : INT := 31;
	out_min : REAL;
	out_max : REAL := 10.0;
	code_min : DWORD;
	code_max : DWORD := 16#FFFFFFFF;
	error_output : REAL;
	overflow_output : REAL := 10.0;
END_VAR
VAR_OUTPUT
	out : REAL;
	sign : BOOL;
	error : BOOL;
	overflow : BOOL;
END_VAR
VAR
	tB: DWORD;
END_VAR

(*
version 1.3	10. mar. 2009
programmer 	oscat
tested by		tobias

Ain1 converts signals from A/D converters or other digital sources to an internal real value.

*)

(* extract error bit *)
error := ((SHR(in,error_bit) AND 16#0000_0001) = 1) OR (error_code_en AND error_code = in);
IF error THEN
	out := error_output;
	RETURN;
END_IF;

(* strip off the data input *)
tb := SHR(SHL(in, 31 - bit_N), 31 - bit_N + Bit_0);

(* extract overflow bit *)
overflow := ((SHR(in,overflow_bit) AND 16#0000_0001) = 1) OR (overflow_code_en AND overflow_code = in) OR (tb < code_min OR tb > code_max);
IF overflow THEN
	out := overflow_output;
	RETURN;
END_IF;

(* extract sign bit *)
sign := (SHR(in,sign_bit) AND 16#0000_0001) = 1;

(* convert in to out *)
out := (DWORD_TO_REAL(tb - code_min) * (out_max - out_min) / DWORD_TO_REAL(code_max - code_min) + out_min);
IF sign THEN out := out * -1.0; END_IF;



(* revision history
hm	23. feb 2008	rev 1.0
	original version

hm	16. mar 2008	rev 1.1
	added type conversions to avoid warnngs under codesys 30

hm	22. apr. 2008	rev 1.2
	corrected error in formula when code_min was set
	corrected error when sign bit was used
	optimized code for better performance

hm	10. mar. 2009	rev 1.3
	real constants updated to new systax using dot

*)

END_FUNCTION_BLOCK

// POUs/Engineering/measurements/ALARM_2
FUNCTION_BLOCK ALARM_2
VAR_INPUT
	X : REAL;
	LO_1 : REAL;
	HI_1 : REAL;
	LO_2 : REAL;
	HI_2 : REAL;
	HYS : REAL;
END_VAR
VAR_OUTPUT
	Q1_LO : BOOL;
	Q1_HI : BOOL;
	Q2_LO : BOOL;
	Q2_HI : BOOL;
END_VAR
VAR
	tmp: REAL;
END_VAR

(*
	version 1.1	11. mar. 2009
	programmer 	hugo
	tested BY		tobias

ALARM_2 will check two pairs of limits and signal when the input is above or below a set limit.
with the input HYS a hysteresis can be defined for all limits. 

*)

tmp := X - Hys * 0.5;
IF tmp > LO_1 THEN Q1_LO := FALSE; END_IF;
IF tmp > LO_2 THEN Q2_LO := FALSE; END_IF;
IF tmp > HI_1 THEN Q1_HI := TRUE; END_IF;
IF tmp > HI_2 THEN Q2_HI := TRUE; END_IF;
tmp := tmp + hys;
IF tmp < LO_1 THEN Q1_LO := TRUE; END_IF;
IF tmp < LO_2 THEN Q2_LO := TRUE; END_IF;
IF tmp < HI_1 THEN Q1_HI := FALSE; END_IF;
IF tmp < HI_2 THEN Q2_HI := FALSE; END_IF;



(* revision history
hm	19. may. 2008		rev 1.0
	original version

hm	11. mar. 2009	rev 1.1
	improved code
*)

END_FUNCTION_BLOCK

// POUs/Engineering/signal processing/AOUT
FUNCTION AOUT : DWORD
VAR_INPUT
	in : REAL;
END_VAR
VAR_INPUT CONSTANT
	Bits : BYTE;
	sign : BYTE := 255;
	low : REAL;
	high : REAL := 10.0;
END_VAR
VAR CONSTANT
	ff : DWORD := 2#1;
END_VAR
VAR
	in2 : REAL;
	sx : BOOL;
END_VAR

(*
version 1.4	23 feb 2008
programmer 	oscat
tested by		tobias

this module conditions an internal real value for D/A converter.
Aout converts and internal real value to a word for an D/A converter or other output devices.
The input value is converted to a n-bit wide output and a sign bit is set separately as specified.
the outout min value is set for the specified min input value and the max output is set for the max input value.
an input higher or lower then the max or min value will set the respective max or min value or the output.


*)

(* if sign bit is defined *)
IF sign < 32 THEN
	sx := sign_R(in);
	in2 := ABS(in);
ELSE
	in2 := in;
END_IF;

(* begrenze in auf die zulässigen werte *)
in2 := LIMIT(low, in2, high);

(* Berechne den Ausgangswert *)
Aout := REAL_TO_DWORD((in2 - low) / (high - low) * DWORD_TO_REAL(SHL(ff,bits) -1));
IF sx THEN Aout := SHL(ff,sign) OR Aout; END_IF;

(*
revision history

hm 18.1.2007		rev 1.1
	renamed Modul to aout.
	changed Output to 32 Bit max.
	corrected error with sign bit.

hm	13.9.2007		rev 1.2
	changed code to avoid warning under codesys 2.8.1

hm	2. dec 2007		rev 1.3
	changed code for better performance

hm	23. feb 2008	rev 1.4
	changed code for better performance
*)

END_FUNCTION

// POUs/Mathematical/SIGN_R
FUNCTION SIGN_R : BOOL
VAR_INPUT
	in : REAL;
END_VAR


(*
version 1.4	10. mar. 2009
programmer 	hugo
tested by		tobias

this function return true if the real input is negative

*)

SIGN_R := in < 0.0;


(* revision history
hm 19.1.2007	rev 1.1
	changed method of function for better compatibility to other systems

hm	1.12.2007	rev 1.2
	changed code to improve performance

hm	14. jun. 2008	rev 1.3
	improved performace

hm 10. mar. 2009	rev 1.4
	real constants updated to new systax using dot																																																																																																																																																																																																																																																																																																																																																																																																																																																																																																																																																																																																																																																																																																																																																																																																																																																																																																																																																																																																																																																											

*)

END_FUNCTION

// POUs/Engineering/signal processing/AOUT1
FUNCTION AOUT1 : DWORD
VAR_INPUT
	in : REAL;
END_VAR
VAR_INPUT CONSTANT
	Bit_0 : INT;
	Bit_N : INT := 31;
	sign : INT := 255;
	low : REAL;
	high : REAL := 10.0;
END_VAR
VAR CONSTANT
	ff : DWORD := 2#1;
END_VAR
VAR
	sx: BOOL;
	in2 : REAL;
END_VAR

(*
version 1.0	23 feb 2008
programmer 	oscat
tested by		tobias

this module conditions an internal real value for a D/A converter.

*)

(* if sign bit is defined *)
IF sign < 32 THEN
	sx := SIGN_R(in);
	in2 := ABS(in);
ELSE
	in2 := in;
END_IF;

(* begrenze in auf die zulässigen werte *)
in2 := LIMIT(low, in2, high);

(* Berechne den Ausgangswert *)
AOUT1 := SHL(REAL_TO_DWORD((in2 - low) / (high - low) * DWORD_TO_REAL(SHL(ff,bit_n - Bit_0 + 1) -1)),Bit_0);
IF sx THEN AOUT1 := SHL(ff,sign) OR AOUT1; END_IF;


(* revision history
hm	23. feb 2008	rev 1.0
	original version

*)

END_FUNCTION

// POUs/Mathematical/Array/ARRAY_GAV
FUNCTION ARRAY_GAV : REAL
VAR_INPUT
	pt : POINTER TO ARRAY[0..32000] OF REAL;
	size : UINT;
END_VAR
VAR
	i: UINT;
	stop: UINT;
END_VAR

(*
version 1.1	10. mar. 2009
programmer 	hugo
tested by		tobias

this function will calculate the geometric average of a given array.
the function needs to be called:	array_avg(adr("array"),sizeof("array"));
because this function works with pointers its very time efficient and it needs no extra memory.

*)

stop := SHR(size,2)-1;
ARRAY_GAV := 1.0;
FOR i := 0 TO stop DO
	IF pt^[i] > 0.0 THEN
		ARRAY_GAV := ARRAY_GAV * pt^[i];
	ELSE
		ARRAY_GAV := 0.0;
		RETURN;
	END_IF;
END_FOR;
ARRAY_GAV := SQRTN(ARRAY_GAV,UINT_TO_INT(stop)+1);


(* revision history
hm	2. apr 2008	rev 1.0
	original version

hm	10. mar. 2009	rev 1.1
	real constants updated to new systax using dot

*)

END_FUNCTION

// POUs/Mathematical/SQRTN
FUNCTION SQRTN : REAL
VAR_INPUT
	X : REAL;
	N : INT;
END_VAR


(*
version 1.3	10. mar. 2009
programmer 	hugo
tested by		tobias

this function calculates the nth root function of X according to the formula sqrtn = x^(1/n).

*)

IF N > 0 THEN
	SQRTN := EXP(LN(x) / INT_TO_REAL(n));
ELSE
	SQRTN := 0.0;
END_IF;


(* revision history
hm		12 jan 2007	rev 1.0
	original version

hm		2. dec 2007	rev 1.1
	changed code for better performance

hm		11. mar 2008	rev 1.2
	added result 0 for compatibility reasons

hm 10. mar. 2009	rev 1.3
	added type conversions for compatibility reasons																																																																																																																																																																																																																																																																																																																																																																																																																																																																																																																																																																																																																																																																																																																																																																																																																																																																																																																																																																																																																																																									

*)

END_FUNCTION

// POUs/Mathematical/Array/ARRAY_HAV
FUNCTION ARRAY_HAV : REAL
VAR_INPUT
	pt : POINTER TO ARRAY[0..32000] OF REAL;
	size : UINT;
END_VAR
VAR
	i: UINT;
	stop: UINT;
END_VAR

(*
version 1.1	10. mar. 2009
programmer 	hugo
tested by		tobias

this function will calculate the harmonic average of a given array.
the function needs to be called:	array_avg(adr("array"),sizeof("array"));
because this function works with pointers its very time efficient and it needs no extra memory.

*)

stop := SHR(size,2)-1;
FOR i := 0 TO stop DO
	IF pt^[i] <> 0.0 THEN
		ARRAY_HAV := ARRAY_HAV + 1.0 / pt^[i];
	ELSE
		ARRAY_HAV := 0.0;
		RETURN;
	END_IF;
END_FOR;
ARRAY_HAV := UINT_TO_REAL(stop + 1) / ARRAY_HAV;


(* revision history
hm	2. apr 2008	rev 1.0
	original version

hm	10. mar. 2009	rev 1.1
	real constants updated to new systax using dot

*)

END_FUNCTION

// POUs/Mathematical/Array/ARRAY_MAX
FUNCTION ARRAY_MAX : REAL
VAR_INPUT
	pt : POINTER TO ARRAY[0..32000] OF REAL;
	size : UINT;
END_VAR
VAR
	i: UINT;
	stop: UINT;
END_VAR

(*
version 1.1	16. mar. 2008
programmer 	hugo
tested by		tobias

this function will calculate the max value of a given array.
the function needs to be called:	array_max(adr("array"),sizeof("array"));
because this function works with pointers its very time efficient and it needs no extra memory.

*)

stop := (size -SIZEOF(pt)) / SIZEOF(pt);
array_max := pt^[0];
FOR i := 1 TO stop DO
	IF pt^[i] > array_max THEN array_max := pt^[i]; END_IF;
END_FOR;

(* revision history
hm	2. oct 2006		rev 1.0
	original version

hm	16. mar. 2008	rev 1.1
	changed input size to uint
*)

END_FUNCTION

// POUs/Mathematical/Array/ARRAY_MIN
FUNCTION ARRAY_MIN : REAL
VAR_INPUT
	pt : POINTER TO ARRAY[0..32000] OF REAL;
	size : UINT;
END_VAR
VAR
	i: UINT;
	stop: UINT;
END_VAR

(*
version 1.1	16. mar. 2008
programmer 	hugo
tested by		tobias

this function will calculate the min value of a given array.
the function needs to be called:	array_min(adr("array"),sizeof("array"));
because this function works with pointers its very time efficient and it needs no extra memory.

*)

stop := (size - SIZEOF(pt)) / SIZEOF(pt);
array_min := pt^[0];
FOR i := 1 TO stop DO
	IF pt^[i] < array_min THEN array_min := pt^[i]; END_IF;
END_FOR;


(* revision history
hm		2. oct. 2006
	original version

hm		16. mar. 2008
	changed type of input size to uint

*)

END_FUNCTION

// POUs/Mathematical/Array/ARRAY_SDV
FUNCTION ARRAY_SDV : REAL
VAR_INPUT
	pt : POINTER TO ARRAY[0..32000] OF REAL;
	size : UINT;
END_VAR


(*
version 1.1	16. mar 2008
programmer 	hugo
tested by		tobias

this function will calculate the standard deviation of a given array.
the function needs to be called:	array_sdv(adr("array"),sizeof("array"));
because this function works with pointers its very time efficient and it needs no extra memory.

*)

(* standard deviation is simply the square root of the variance *)

array_sdv := SQRT(array_var(pt, size));

(* revision history
hm 	1.4.2007		rev 1.0
	function created

hm	16. mar. 2008	rev 1.1
	changed type of input size to uint

*)

END_FUNCTION

// POUs/Mathematical/Array/ARRAY_VAR
FUNCTION ARRAY_VAR : REAL
VAR_INPUT
	pt : POINTER TO ARRAY[0..32000] OF REAL;
	size : UINT;
END_VAR
VAR
	avg : REAL;
	i: UINT;
	stop: UINT;
END_VAR

(*
version 1.3	10. mar. 2009
programmer 	hugo
tested by		tobias

this function will calculate the variance of a given array.
the function needs to be called:	array_var(adr("array"),sizeof("array"));
because this function works with pointers its very time efficient and it needs no extra memory.

*)

(* at first we calualte the arithmetic average of the array *)

stop := SHR(size,2)-1;
avg := pt^[0];
FOR i := 1 TO stop DO
	avg := avg + pt^[i];
END_FOR;
avg := avg / UINT_TO_REAL(stop + 1);

(* in a second run we calculate the variance of the array *)

array_var := (pt^[0] - avg) * (pt^[0] - avg);
FOR i := 1 TO stop DO
	array_var := array_var + (pt^[i] - avg) * (pt^[i] - avg);
END_FOR;
ARRAY_VAR := ARRAY_VAR / UINT_TO_REAL(stop);

(* revision history
hm 	1.4.2007	rev 1.0
	function created

hm	12.12.2007	rev 1.1
	changed code for better performance

hm	16. mar. 2008	rev 1.2
	changed type of input size to uint

hm	10. mar. 2009	rev 1.3
	added type conversions for compatibility reasons
*)

END_FUNCTION

// POUs/Time&Date/SECOND
FUNCTION SECOND : REAL
VAR_INPUT
	itod : TOD;
END_VAR


(*
version 1.1	2 oct 2006
programmer 	hugo
tested by	oscat

returns the seconds and milliseconds as real of TOD   
 
*)

SECOND := DWORD_TO_REAL(TOD_TO_DWORD(itod) - TOD_TO_DWORD(itod)/60000 * 60000) / 1000.0;



(* change history

hm	2. oct. 2006 rev 1.1 
	changed name of input to itod

*)

END_FUNCTION

// POUs/Mathematical/Array/ARRAY_SPR
FUNCTION ARRAY_SPR : REAL
VAR_INPUT
	pt : POINTER TO ARRAY[0..32000] OF REAL;
	size : UINT;
END_VAR
VAR
	i: UINT;
	stop: UINT;
	array_max : REAL;
	array_min : REAL;
END_VAR

(*
version 1.1	16. mar. 2008
programmer 	hugo
tested by		tobias

this function will calculate the spread of a given array.
the function needs to be called:	array_spr(adr("array"),sizeof("array"));
for example: spread of [12,0,4,1,7] is 12 - 0 = 12.
because this function works with pointers its very time efficient and it needs no extra memory.

*)

stop := (size -SIZEOF(pt)) / SIZEOF(pt);
array_min := pt^[0];
array_max := pt^[0];
FOR i := 1 TO stop DO
	IF pt^[i] > array_max THEN array_max := pt^[i];
	ELSIF pt^[i] < array_min THEN array_min := pt^[i];
	END_IF;
END_FOR;
array_spr := array_max - array_min;


(* revision history
hm 	2. oct. 2006	rev 1.0
	original version

hm	16. mar. 2008	rev 1.1
	changed type of input size to uint

*)

END_FUNCTION

// POUs/Mathematical/Array/ARRAY_SUM
FUNCTION ARRAY_SUM : REAL
VAR_INPUT
	pt : POINTER TO ARRAY[0..32000] OF REAL;
	size : UINT;
END_VAR
VAR
	i: UINT;
	stop: UINT;
END_VAR


(*
version 1.1	16. mar. 2008
programmer 	hugo
tested by		tobias

this function will calculate the sum of a given array.
the function needs to be called:	array_sum(adr("array"),sizeof("array"));
because this function works with pointers its very time efficient and it needs no extra memory.

*)

stop := (size -SIZEOF(pt)) / SIZEOF(pt);
array_sum := pt^[0];
FOR i := 1 TO stop DO
	array_sum := array_sum + pt^[i];
END_FOR;

(* revision history
hm 	2. oct. 2006	rev 1.0
	function created

hm	16. mar. 2008	rev 1.1
	changed type of input size to uint

*)

END_FUNCTION

// POUs/Mathematical/Array/ARRAY_TREND
FUNCTION ARRAY_TREND : REAL
VAR_INPUT
	pt : POINTER TO ARRAY[0..32000] OF REAL;
	size : UINT;
END_VAR
VAR
	i: UINT;
	stop: UINT;
	x: REAL;
	stop2: UINT;
END_VAR

(*
version 1.3	10. mar. 2009
programmer 	hugo
tested by		tobias

this function will calculate the trend of a given array.
trend will calculate the avg of the first half of the array and then the avg of the second half, trend = avg2 - avg1.
for example:  [0,1,4,5,3,4,6,3] = 4 - 2.5 = 1.5
the function needs to be called:	array_trend(adr("array"),sizeof("array"));
because this function works with pointers its very time efficient and it needs no extra memory.

*)

stop := SHR(size,2)-1;
stop2 := SHR(stop,1);
FOR i := 0 TO stop2 DO x := x - pt^[i]; END_FOR;
IF EVEN(UINT_TO_INT(stop)) THEN
	FOR i := stop2 TO stop DO X := X + pt^[i]; END_FOR;
ELSE
	FOR i := stop2 + 1 TO stop DO X := X + pt^[i]; END_FOR;
END_IF;
ARRAY_TREND := x / UINT_TO_REAL(stop2 + 1);

(* revision history
hm	2 oct 2007	rev 1.0
	original version

hm	12 dec 2007	rev 1.1
	changed code for better performance

hm	16. mar. 2008	rev 1.2
	changed type of input size to uint

hm	10. mar. 2009	rev 1.3
	added type conversions for compatibility reasons
*)

END_FUNCTION

// POUs/Mathematical/ASINH
FUNCTION ASINH : REAL
VAR_INPUT
	X : REAL;
END_VAR


(*
version 1.3	10. mar 2009
programmer 	hugo
tested by		tobias

this function calculates the arcus sin hyperbolicus

*)

ASINH := LN(SQRT(X * X + 1.0)+X);

(* revision history
hm		12 jan 2007	rev 1.0
	original version

hm		2. dec 2007	rev 1.1
	changed code for better performance

hm		16.3. 2007		rev 1.2
	changed sequence of calculations to improve performance

hm	10. mar. 2009		rev 1.3
	real constants updated to new systax using dot

*)

END_FUNCTION

// POUs/Engineering/conversion/ASTRO
FUNCTION_BLOCK ASTRO
VAR_INPUT
	m : REAL;
	AE : REAL;
	PC : REAL;
	LJ : REAL;
END_VAR
VAR_OUTPUT
	Ym : REAL;
	YAE : REAL;
	YPC : REAL;
	YLJ : REAL;
END_VAR


(*
version 1.1	11. mar. 2009
programmer 	hugo
tested by		oscat

this function converts different length units
any unused input can simply be left open.
different inputs connected at the same time will be added up.

*)

YAE :=	AE
		+ m * 6.6845871535E-012
		+ PC * 206265.0
		+ LJ * 63240.0;
Ym := YAE * 149.597870E9;
YPC := YAE * 4.8481322570E-006;
YLJ := YAE * 1.5812776724E-005;


(*
Länge Meter m SI-Basiseinheit
Astronomische Einheit* AE 1 AE = 149,597 870 · E9 m
Parsec pc 1 pc = 206265 AE = 30,857 · E15 m
Lichtjahr Lj 1 Lj = 9,460 530 · E15 m = 63240 AE = 0,306 59 pc
Ångström Å 1 Å = E–l0 m
typograph. Punkt p 1 p = 0,376 065 mm • im Druckereigewerbe
inch** in 1 in = 2,54 · E–2 m = 25,4 mm***
foot ft 1 ft = 0,3048 m = 30,48 cm
yard yd 1 yd = 0,9144 m
mile mile 1 mile = 1609,344 m
Internat. Seemeile sm 1 sm = 1852 m
Fathom fm 1 fm = 1,829 m • in der Seeschifffahrt
*)

(* revision history

hm	27. mar. 2007	rev 1.0
	original version

hm	11. mar. 2009	rev 1.1
	improved code

*)

END_FUNCTION_BLOCK

// POUs/Engineering/conversion/LENGTH
FUNCTION_BLOCK LENGTH
VAR_INPUT
	m : REAL;
	p : REAL;
	in : REAL;
	ft : REAL;
	yd : REAL;
	mile : REAL;
	sm : REAL;
	fm : REAL;
END_VAR
VAR_OUTPUT
	Ym : REAL;
	Yp : REAL;
	Yin : REAL;
	Yft : REAL;
	Yyd : REAL;
	Ymile : REAL;
	Ysm : REAL;
	Yfm : REAL;
END_VAR


(*
version 1.1	11. mar. 2009
programmer 	hugo
tested by		oscat

this function converts different length units
any unused input can simply be left open.
different inputs connected at the same time will be added up.

*)

Ym :=	m
		+ p * 0.000376065
		+ in * 0.0254
		+ ft * 0.3048
		+ yd * 0.9144
		+ mile * 1609.344
		+ sm * 1852.0
		+ fm * 1.829;
Yp := Ym * 2659.11478068951;
Yin := Ym * 39.37007874016;
Yft := Ym * 3.28083989501;
Yyd := Ym * 1.09361329834;
Ymile := Ym * 0.00062137119;
Ysm := Ym * 0.00053995680;
Yfm := Ym * 0.54674685621;

(*
Länge Meter m SI-Basiseinheit
Astronomische Einheit* AE 1 AE = 149,597 870 · E9 m
Parsec pc 1 pc = 206265 AE = 30,857 · E15 m
Lichtjahr Lj 1 Lj = 9,460 530 · E15 m = 63240 AE = 0,306 59 pc
Ångström Å 1 Å = E–l0 m
typograph. Punkt p 1 p = 0,376 065 mm • im Druckereigewerbe
inch** in 1 in = 2,54 · E–2 m = 25,4 mm***
foot ft 1 ft = 0,3048 m = 30,48 cm
yard yd 1 yd = 0,9144 m
mile mile 1 mile = 1609,344 m
Internat. Seemeile sm 1 sm = 1852 m
Fathom fm 1 fm = 1,829 m • in der Seeschifffahrt
*)

(* revision history

hm	27. mar. 2007	rev 1.0
	original version

hm	11. mar. 2009	rev 1.1
	improved code

*)

END_FUNCTION_BLOCK

// POUs/Mathematical/ATAN2
FUNCTION ATAN2 : REAL
VAR_INPUT
	Y : REAL;
	X : REAL;
END_VAR


(*
version 1.2	10. mar. 2009
programmer 	hugo
tested by		oscat

this function calculates the angle in a coordinate system in rad.

*)

IF X > 0.0 THEN
	ATAN2 := ATAN(Y/X);
ELSIF X < 0.0 THEN
	IF Y >=0.0 THEN
		ATAN2 := ATAN(Y/X) + MATH.PI;
	ELSE
		ATAN2 := ATAN(Y/X) - MATH.PI;
	END_IF;
ELSIF Y > 0.0 THEN
	ATAN2 := MATH.PI05;
ELSIF Y < 0.0 THEN
	ATAN2 := -MATH.PI05;
ELSE
	ATAN2 := 0.0;
END_IF;


(* revision history
hm	20.  apr. 2008	rev 1.0
	original version

hm	18. oct. 2008	rev 1.1
	changed to use math constants

hm	10. mar. 2009	rev 1.2
	real constants updated to new systax using dot

*)

END_FUNCTION

// POUs/Mathematical/RAD
FUNCTION RAD : REAL
VAR_INPUT
	DEG : REAL;
END_VAR


(*
version 1.2	18. oct. 2008
programmer 	hugo
tested by	tobias

this function converts Radiant to degrees

*)

RAD := MODR(0.0174532925199433 * DEG, math.PI2);

(* revision history
hm	4. aug 2006		rev 1.0
	original version

hm 	16. oct 2007	rev 1.1
	added modr statement which prohibits rad to become bigger than 2PI

hm	18. oct 2008	rev 1.2
	using math constants

*)

END_FUNCTION

// POUs/Mathematical/DEG
FUNCTION DEG : REAL
VAR_INPUT
	rad : REAL;
END_VAR


(*
version 1.2	10. mar. 2009
programmer 	hugo
tested by		tobias

this function converts degrees into Radiant
execution time on wago 750 - 841 =  10  us
*)

DEG := MODR(57.29577951308232 * RAD, 360.0);

(* revision history
hm	4. aug 2006	rev 1.0
	original version

hm 16. oct 2007	rev 1.1
	added modr statement which prohibits deg to become bigger than 360

hm	10. mar. 2009	rev 1.2
	real constants updated to new systax using dot
*)

END_FUNCTION

// POUs/Mathematical/ATANH
FUNCTION ATANH : REAL
VAR_INPUT
	X : REAL;
END_VAR


(*
version 1.2	10. mar. 2009
programmer 	hugo
tested by		tobias

this function calculates the arcus tangens hyperbolicus

*)

ATANH := LN((1.0 + x)/(1.0 - x)) * 0.5;


(* revision history
hm		12 jan 2007	rev 1.0
	original version

hm		5. jan 2008	rev 1.1
	improved code for better performance

hm	10. mar. 2009		rev 1.2
	real constants updated to new systax using dot

*)

END_FUNCTION

// POUs/Logic/generators/B_TRIG
FUNCTION_BLOCK B_TRIG
VAR_INPUT
	CLK : BOOL;
END_VAR
VAR_OUTPUT
	Q : BOOL;
END_VAR
VAR
	edge : BOOL;
END_VAR

(*
version 1.0	4. aug. 2006
programmer 	hugo
tested by		tobias

this block is similar to R_trig and F_trig but it generates a pulse on rising and falling edge.

*)

Q := clk XOR edge;
edge := CLK;


(* revision history
hm		4. aug. 2006	rev 1.0
	original version

*)

END_FUNCTION_BLOCK

// POUs/Engineering/control/BAND_B
FUNCTION BAND_B : BYTE
VAR_INPUT
	X : BYTE;
	B : BYTE;
END_VAR



(*
version 1.0	21. Nov. 2008
programmer 	hugo
tested by	oscat

BAND_B will limit X to B <= X <= 255-B. while X < B the resulkt will be 0 and while X > 255-B the output will be 255
otherwise the result = X.

*)

IF X < B THEN
	BAND_B := 0;
ELSIF X > BYTE#255-B THEN
	BAND_B := 255;
ELSE
	BAND_B := X;
END_IF;



(* revision history
hm	21. nov. 2008	rev 1.0
	original version

*)

END_FUNCTION

// POUs/Engineering/measurements/BAR_GRAPH
FUNCTION_BLOCK BAR_GRAPH
VAR_INPUT
	X : REAL;
	rst : BOOL;
END_VAR
VAR_INPUT CONSTANT
	trigger_Low : REAL;
	trigger_High : REAL;
	Alarm_low : BOOL;
	Alarm_high : BOOL;
	log_scale : BOOL;
END_VAR
VAR_OUTPUT
	LOW, Q1, Q2, Q3, Q4, Q5, Q6, HIGH : BOOL;
	Alarm : BOOL;
	Status : BYTE;
END_VAR
VAR
	init : BOOL;
	T1, T2, T3, T4, T5 : REAL;
END_VAR
VAR
	temp : REAL;
END_VAR

